// ----------------------------------------------------------
// LI_S Säuretank
// ----------------------------------------------------------
      L     DB1821.DBD 1118; // !!! insert correct SFM !!!
      T     DB2823.DBD  238;

//      SET
//      =     "U082AnID".LI_S.EAlHH

// ----------------------------------------------------------
// CS_S Säuretank
// ----------------------------------------------------------
      L     DB1821.DBD 1118; // !!! insert correct SFM !!!
      T     DB2823.DBD  358;

      SET   ;
      =     DB2823.DBX  261.5;

NETWORK
TITLE =Universal Value

      NOP   0;

// ----------------------------------------------------------
// unv001 Process Status
// ----------------------------------------------------------
// process value to UnV
//      L     0.000000e+000
//      T     "U082UnVD".unv001.ValExt

// ----------------------------------------------------------
// unv002 Universal Value 02
// ----------------------------------------------------------
// process value to UnV
//      L     0.000000e+000
//      T     "U082UnVD".unv002.ValExt

NETWORK
TITLE =Special Input

      NOP   0;

// ----------------------------------------------------------
// LS_LLL_SAEURE Säuretank LS-
// ----------------------------------------------------------
      ON    DB2910.DBX  582.5;
      ON    DB2920.DBX  582.5;
      ON    DB2930.DBX  582.5;
      =     DB2821.DBX   81.4;
      CLR   ;
      =     DB2821.DBX   81.5;

// ----------------------------------------------------------
// LS_HL_SAEURE Säuretank LS+
// ----------------------------------------------------------
      ON    DB2910.DBX  822.5;
      ON    DB2920.DBX  822.5;
      ON    DB2930.DBX  822.5;
      =     DB2821.DBX  141.4;
      SET   ;
      =     DB2821.DBX  141.5;

      SET   ;
      =     DB2821.DBX  140.6;

// ----------------------------------------------------------
// LS_LL_SAEURE Säuretank LS/
// ----------------------------------------------------------
      CLR   ;
//      =     "U082SpID".LS_LL_SAEURE.EAl
      =     DB2821.DBX  201.5;

// ----------------------------------------------------------
// LS_LL_SAEURE_ALT
// ----------------------------------------------------------
      SET   ;
      =     DB2821.DBX  261.4;
      =     DB2821.DBX  261.5;

// ----------------------------------------------------------
// LANG_NEUANSATZ_SAEURE RUECKMELDUNG VON LANG AN TU
// ----------------------------------------------------------
      CLR   ;
//      =     "U082SpID".LANG_NEUANSATZ_SAEURE.EAl
//     =     "U082SpID".LANG_NEUANSATZ_SAEURE.Pre

// ----------------------------------------------------------
// LANG_NACHSCH_SAEURE RUECKMELDUNG VON LANG AN TU
// ----------------------------------------------------------
      CLR   ;
//      =     "U082SpID".LANG_NACHSCH_SAEURE.EAl
//      =     "U082SpID".LANG_NACHSCH_SAEURE.Pre

NETWORK
TITLE =Messages

      NOP   0;

// ----------------------------------------------------------
// msg001 Message 01
// ----------------------------------------------------------
      SET   ;
      R     DB2827.DBX   80.7;
      =     DB2827.DBX   81.4;

      CLR   ;
      =     DB2827.DBX   82.7;

// ----------------------------------------------------------
// msg002 Message 02
// ----------------------------------------------------------
      SET   ;
      R     DB2827.DBX  140.7;
      =     DB2827.DBX  141.4;

      CLR   ;
      =     DB2827.DBX  142.7;

NETWORK
TITLE =Sequence organisation

      CLR   ;
      =     M    122.2;

// SFM supply ----------------------------------------------------------------

// analog value to SFM Säuretank -----------------------
      L     DB2823.DBD  146;
      T     DB1821.DBD  386; // Level

// analog value to SFM Säuretank -----------------------
      L     DB2823.DBD  266;
      T     DB1821.DBD  642; // Conductivity
      T     DB1821.DBD  658; // Conductivity Start Pulse/Pause

// sequencer ----------------------------------------------------------------
      A     DB1823.DBX   43.1;
      S     DB1823.DBX   97.3;

      CALL FC    40 (
           UnitNo                   := #UnitNo);

NETWORK
TITLE =Auto / Manual

      SET   ;
      AN    M    122.2;
      JC    MODE;
      AN    M    120.1;

// assign actuator mode
      AN    M    120.1;
      =     DB2820.DBX  105.4;
      =     DB2820.DBX  185.4;
      =     DB2820.DBX  345.4;
      =     DB2820.DBX  425.4;
      =     DB2820.DBX  585.4;
      =     DB2820.DBX  665.4;
      =     DB2820.DBX  745.4;



MODE: SET   ;

NETWORK
TITLE =RW_SAEURE Rührwerk S1T
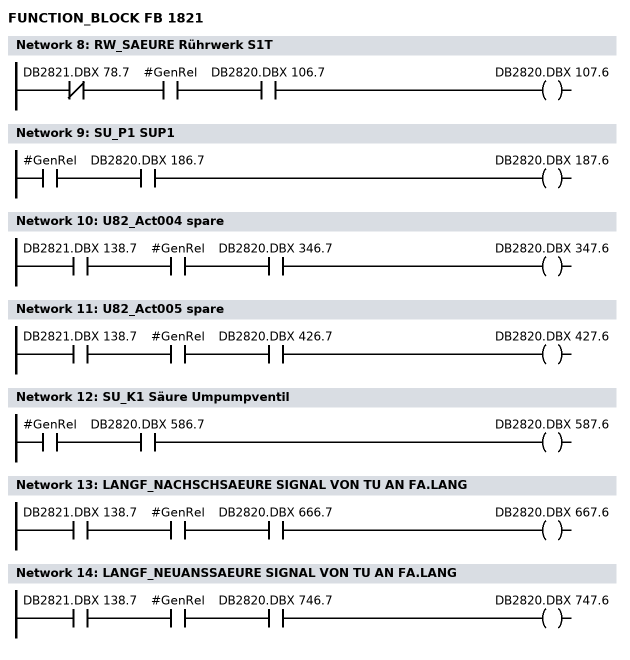

      AN    DB2821.DBX   78.7;
      A     #GenRel;
      A     DB2820.DBX  106.7;
      =     DB2820.DBX  107.6;
NETWORK
TITLE =SU_P1 SUP1

      A     #GenRel;
      A     DB2820.DBX  186.7;
      =     DB2820.DBX  187.6;
NETWORK
TITLE =U82_Act004 spare

      A     DB2821.DBX  138.7;

      A     #GenRel;
      A     DB2820.DBX  346.7;
      =     DB2820.DBX  347.6;
NETWORK
TITLE =U82_Act005 spare

      A     DB2821.DBX  138.7;

      A     #GenRel;
      A     DB2820.DBX  426.7;
      =     DB2820.DBX  427.6;
NETWORK
TITLE =SU_K1 Säure Umpumpventil

      A     #GenRel;
      A     DB2820.DBX  586.7;
      =     DB2820.DBX  587.6;
NETWORK
TITLE =LANGF_NACHSCHSAEURE SIGNAL VON TU AN FA.LANG

      A     DB2821.DBX  138.7;

      A     #GenRel;
      A     DB2820.DBX  666.7;
      =     DB2820.DBX  667.6;
NETWORK
TITLE =LANGF_NEUANSSAEURE SIGNAL VON TU AN FA.LANG

      A     DB2821.DBX  138.7;

      A     #GenRel;
      A     DB2820.DBX  746.7;
      =     DB2820.DBX  747.6;
END_FUNCTION_BLOCK

FUNCTION_BLOCK FB 1830
TITLE =U083: Hot Water Tank
FAMILY : BOTEC_F1
NAME : UniA
VERSION : 2.1


VAR_TEMP
  EStopOK : BOOL ;	//auxiliary flag
  CIP : BOOL ;	//CIP Program Selected
  xTmp : BOOL ;	//Temporary Bool(free for general use)
  UnitNo : INT ;	//unit number
  UnitFB : INT ;	//unit expansion FB number
  rTmp : REAL ;	//Temporary REAL (free for general use)
  iTmp : INT ;	//Temporary INT (free for general use)
  dTmp : DINT ;	//Temporary DINT (free for general use)
END_VAR
BEGIN
NETWORK
TITLE =general

      CLR   ;
      =     #xTmp;
      =     #EStopOK;

      L     DB1830.DBW    0;
      T     #UnitNo;
      L     DB1830.DBW    2;
      T     #UnitFB;

NETWORK
TITLE =analog inputs

      NOP   0;
// LI_HW AnI 001 Niveau Heisswassertank
      CALL FC    24 (
           UnitNo                   := #UnitNo,
           AnIRec                   := DB2833.LI_HW,
           ValPer                   := IW   534);

// HWT_TT01 AnI 002 Temp. HWT
      CALL FC    24 (
           UnitNo                   := #UnitNo,
           AnIRec                   := DB2833.HWT_TT01,
           ValPer                   := IW   536);

// HWT_PIC02 AnI 003
      CALL FC    24 (
           UnitNo                   := #UnitNo,
           AnIRec                   := DB2833.HWT_PIC02,
           ValPer                   := IW   542);

// U83_AnI004 AnI 004 spare
      CALL FC    24 (
           UnitNo                   := #UnitNo,
           AnIRec                   := DB2833.U83_AnI004,
           ValPer                   := IW   236);

// HWT_TT02 AnI 005 Temp. nach Ausdehnungsgefaess
      CALL FC    24 (
           UnitNo                   := #UnitNo,
           AnIRec                   := DB2833.HWT_TT02,
           ValPer                   := IW   538);

// HWT_FT01 AnI 006
      CALL FC    24 (
           UnitNo                   := #UnitNo,
           AnIRec                   := DB2833.HWT_FT01,
           ValPer                   := IW   544);

NETWORK
TITLE =Universal value

      NOP   0;
// unv001 UnV 001 Process Status
      CALL FC    27 (
           UnitNo                   := #UnitNo,
           UnVRec                   := DB2835.unv001,
           ValExt                   := DB2835.DBD  234);

// unv002 UnV 002 Universal Value 02
      CALL FC    27 (
           UnitNo                   := #UnitNo,
           UnVRec                   := DB2835.unv002,
           ValExt                   := DB2835.DBD  362);

NETWORK
TITLE =special inputs

      NOP   0;
// LS_LL_HWT SpI 001 Heißwassertank LS-
      CALL FC    14 (
           UnitNo                   := #UnitNo,
           SpIRec                   := DB2831.LS_LL_HWT,
           SpIBit                   := I     93.4);

// LS_HL_HWT SpI 002 Heißwassertank LS+
      CALL FC    14 (
           UnitNo                   := #UnitNo,
           SpIRec                   := DB2831.LS_HL_HWT,
           SpIBit                   := I     93.2);

// LS_HL_HWA SpI 003 Ausdehnungsgefäß HWT LS+
      CALL FC    14 (
           UnitNo                   := #UnitNo,
           SpIRec                   := DB2831.LS_HL_HWA,
           SpIBit                   := I     93.3);

// SpI4 SpI 004 spare
      CALL FC    14 (
           UnitNo                   := #UnitNo,
           SpIRec                   := DB2831.SpI4,
           SpIBit                   := #xTmp);

// RM_NI_HW_K1 SpI 005
      CALL FC    14 (
           UnitNo                   := #UnitNo,
           SpIRec                   := DB2831.RM_NI_HW_K1,
           SpIBit                   := I     68.4);

// NI_PANEEL_3_NI1 SpI 006 PANEEL3 RV.K2 - HWT
      CALL FC    14 (
           UnitNo                   := #UnitNo,
           SpIRec                   := DB2831.NI_PANEEL_3_NI1,
           SpIBit                   := I     68.0);

// S6_HWP1_HAND_EIN_LAUTO SpI 007 SCHALTER PUMPE HW.P1
      CALL FC    14 (
           UnitNo                   := #UnitNo,
           SpIRec                   := DB2831.S6_HWP1_HAND_EIN_LAUTO,
           SpIBit                   := I     64.3);

NETWORK
TITLE =messages

      NOP   0;
// msg001 Msg 001 Message 01
      CALL FC    16 (
           UnitNo                   := #UnitNo,
           MsgRec                   := DB2837.msg001,
           MsgBit                   := DB2837.DBX   82.7);

// msg002 Msg 002 Message 02
      CALL FC    16 (
           UnitNo                   := #UnitNo,
           MsgRec                   := DB2837.msg002,
           MsgBit                   := DB2837.DBX  142.7);

NETWORK
TITLE =counters

      NOP   0;
// U83_Cnt001 Cnt 001 spare
      CALL FC    25 (
           UnitNo                   := #UnitNo,
           CntRec                   := DB2832.U83_Cnt001,
           Imp                      := DB2832.DBX   99.0);

NETWORK
TITLE =controllers

      NOP   0;
// HWP1_FU PID 001 FU Heisswasserpumpe
      CALL FC    55 (
           UnitNo                   := #UnitNo,
           PIDRec                   := DB2836.HWP1_FU,
           SpExt                    := DB2836.DBD  234,
           PVal                     := DB2836.DBD  254,
           OPer                     := PQW  532);

// RV_Kaltwasser PID 002 Kaltwasser Regelventil HWT
      CALL FC    55 (
           UnitNo                   := #UnitNo,
           PIDRec                   := DB2836.RV_Kaltwasser,
           SpExt                    := DB2836.DBD  414,
           PVal                     := DB2836.DBD  434,
           OPer                     := QW   524);

// U83_PID003 PID 003 spare
      CALL FC    55 (
           UnitNo                   := #UnitNo,
           PIDRec                   := DB2836.U83_PID003,
           SpExt                    := DB2836.DBD  594,
           PVal                     := DB2836.DBD  614,
           OPer                     := QW   232);// S5 ?

NETWORK
TITLE =unit supply

      UC    FB [#UnitFB];

NETWORK
TITLE =HWP1  Heisswasserpumpe Ansteuerung FU
// Act 001
// Box           : LT-CIP
// Input address : I256.5
// Output address: Q256.5
      CALL FC    70 (
           UnitNo                   := #UnitNo,
           ActRec                   := DB2830.HWP1,
           Typ                      := 0,
           FBa                      := #xTmp,
           FBa2                     := #xTmp,
           Out                      := Q    256.5);

NETWORK
TITLE =HWP1_NETZ  Heisswasserpumpe Netzschütz
// Act 002
// Box           : LT-CIP
// Output address: Q256.6
      CALL FC    70 (
           UnitNo                   := #UnitNo,
           ActRec                   := DB2830.HWP1_NETZ,
           Typ                      := 1,
           FBa                      := #xTmp,
           FBa2                     := I    256.5,
           Out                      := Q    256.6);

NETWORK
TITLE =U83_Act003  spare
// Act 003
// Box           :
// Output address: #xTmp
      CALL FC    70 (
           UnitNo                   := #UnitNo,
           ActRec                   := DB2830.U83_Act003,
           Typ                      := 0,
           FBa                      := #xTmp,
           FBa2                     := #xTmp,
           Out                      := #xTmp);

NETWORK
TITLE =U83_Act004  spare
// Act 004
// Box           :
// Output address: #xTmp
      CALL FC    70 (
           UnitNo                   := #UnitNo,
           ActRec                   := DB2830.U83_Act004,
           Typ                      := 0,
           FBa                      := #xTmp,
           FBa2                     := #xTmp,
           Out                      := #xTmp);

NETWORK
TITLE =U83_Act005  spare
// Act 005
// Box           :
// Output address: #xTmp
      CALL FC    70 (
           UnitNo                   := #UnitNo,
           ActRec                   := DB2830.U83_Act005,
           Typ                      := 0,
           FBa                      := #xTmp,
           FBa2                     := #xTmp,
           Out                      := #xTmp);

NETWORK
TITLE =HWT_V1  HWT Abnahmeventil
// Act 007
// Box           : VSRVK1..3
// Input address : I275.6
// Output address: Q275.6
      CALL FC    70 (
           UnitNo                   := #UnitNo,
           ActRec                   := DB2830.HWT_V1,
           Typ                      := 1,
           FBa                      := #xTmp,
           FBa2                     := I    275.6,
           Out                      := Q    275.6);

NETWORK
TITLE =HWT_V2
// Act 009
// Box           : VS-RRA
// Input address : I201.2
// Output address: Q201.2
      CALL FC    70 (
           UnitNo                   := #UnitNo,
           ActRec                   := DB2830.HWT_V2,
           Typ                      := 1,
           FBa                      := #xTmp,
           FBa2                     := I    201.2,
           Out                      := Q    201.2);

NETWORK
TITLE =HWT_V3
// Act 010
// Box           : VS-RRA
// Input address : I201.3
// Output address: Q201.3
      CALL FC    70 (
           UnitNo                   := #UnitNo,
           ActRec                   := DB2830.HWT_V3,
           Typ                      := 1,
           FBa                      := #xTmp,
           FBa2                     := I    201.3,
           Out                      := Q    201.3);

NETWORK
TITLE =HW_WT1_V1  NEU Dampfabsperrung HW-WT1 schließen
// Act 011
// Box           : VSHF9
// Input address : I116.7
// Output address: Q117.0
//      CALL  "Act"
//       UnitNo:=#UnitNo
//       ActRec:="U083ActD".HW_WT1_V1
//       Typ   :=0
//       FBa   :=#xTmp
//       FBa2  :="HW_WT1_V1GSC"
//       Out   :="HW_WT1_V1O"

NETWORK
TITLE =HWT_V4  HWT Luftventil Ausdehnungsgefäß
// Act 012
// Box           : VSRVK1..3
// Input address : I275.7
// Output address: Q275.7
      CALL FC    70 (
           UnitNo                   := #UnitNo,
           ActRec                   := DB2830.HWT_V4,
           Typ                      := 1,
           FBa                      := #xTmp,
           FBa2                     := I    275.7,
           Out                      := Q    275.7);

NETWORK
TITLE =HW_WT1_V1O  NEU Dampfabsperrung HW-WT1 öffnen
// Act 013
// Box           : VSHF9
// Output address: Q116.7

      CALL FC    70 (
           UnitNo                   := #UnitNo,
           ActRec                   := DB2830.HW_WT1_V1O,
           Typ                      := 1,
           FBa                      := #xTmp,
           FBa2                     := I    116.7,
           Out                      := Q    117.0);

END_FUNCTION_BLOCK

FUNCTION_BLOCK FB 1831
TITLE =U083: Hot Water Tank
FAMILY : BOTEC_F1
NAME : UniE
VERSION : 1.2


VAR_TEMP
  CIP : BOOL ;	//CIP active
  UNIM : BOOL ;	//Unit Not In Maintenance
  GenRel : BOOL ;	//general OK (emergency and maintenance OK)
  EStopOK : BOOL ;	//emergency OK
  UnitNo : INT ;	//unit number
  xTmp : BOOL ;	//Temporary Bool
  iTmp : INT ;	//Temporary INT
  rTmp : REAL ;	//Temporary REAL
  dTmp : DINT ;	//Temporary DINT (free for general use)
  RetValInt : INT ;	//return value
END_VAR
BEGIN
NETWORK
TITLE =General

      SET   ;
// Simulation ---------------------------------------------------------------
      A     DB1831.DBX 1357.7;
      CC    FB  1839; // "U083Sim"
      A     DB1831.DBX   17.3;
      =     DB1831.DBX 1357.7; //Help bit for simulation

// get unit number ----------------------------------------------------------
      L     DB1830.DBW    0;
      T     #UnitNo;

// CIP ----------------------------------------------------------------------
      L     DB1831.DBD   54;
      L     0;
      <D    ;
      =     #CIP;

// emergency OK -------------------------------------------------------------
      A     DB1835.DBX   27.0; //Emergency Stop OK
      =     #EStopOK;

// Write Unit in Maintenance ------------------------------------------------

      AN    DB1831.DBX   69.7;
      =     #UNIM;

// emergency and maintenance OK ---------------------------------------------
      A     #EStopOK;
      A     #UNIM;
      =     #GenRel;

// communication ------------------------------------------------------------
      UC    FB  1835; // U083Com

NETWORK
TITLE =Analog Inputs

      NOP   0;

// ----------------------------------------------------------
// LI_HW Niveau Heisswassertank
// ----------------------------------------------------------
      L     DB1831.DBD 1118; // !!! insert correct SFM !!!
      T     DB2833.DBD  238;

//      SET
//      =     "U083AnID".LI_HW.EAlHH

// ----------------------------------------------------------
// HWT_TT01 Temp. HWT
// ----------------------------------------------------------
      L     DB1831.DBD 1118; // !!! insert correct SFM !!!
      T     DB2833.DBD  358;

      SET   ;
      =     DB2833.DBX  261.5;

// ----------------------------------------------------------
// HWT_PIC02
// ----------------------------------------------------------
      L     DB1831.DBD 1118; // !!! insert correct SFM !!!
      T     DB2833.DBD  478;

      SET   ;
      =     DB2833.DBX  381.5;

// ----------------------------------------------------------
// U83_AnI004
// ----------------------------------------------------------
      L     DB1831.DBD 1118; // !!! insert correct SFM !!!
      T     DB2833.DBD  598;

      SET   ;
      =     DB2833.DBX  501.5;

// ----------------------------------------------------------
// HWT_TT02 Temp. nach Ausdehnungsgefaess
// ----------------------------------------------------------
      L     DB1831.DBD 1118; // !!! insert correct SFM !!!
      T     DB2833.DBD  718;

      SET   ;
      =     DB2833.DBX  621.5;

// ----------------------------------------------------------
// HWT_FT01
// ----------------------------------------------------------
      L     DB1831.DBD 1118; // !!! insert correct SFM !!!
      T     DB2833.DBD  838;

      SET   ;
      =     DB2833.DBX  741.5;

NETWORK
TITLE =Universal Value

      NOP   0;

// ----------------------------------------------------------
// unv001 Process Status
// ----------------------------------------------------------
// process value to UnV
//      L     0.000000e+000
//      T     "U083UnVD".unv001.ValExt

// ----------------------------------------------------------
// unv002 Universal Value 02
// ----------------------------------------------------------
// process value to UnV
//      L     0.000000e+000
//      T     "U083UnVD".unv002.ValExt

NETWORK
TITLE =Special Input

      NOP   0;

// ----------------------------------------------------------
// LS_LL_HWT Heißwassertank LS-
// ----------------------------------------------------------
      ON    DB2910.DBX  502.5;
      ON    DB2920.DBX  502.5;
      ON    DB2930.DBX  502.5;
      =     DB2831.DBX   81.4;
      CLR   ;
      =     DB2831.DBX   81.5;

// ----------------------------------------------------------
// LS_HL_HWT Heißwassertank LS+
// ----------------------------------------------------------
      ON    DB2930.DBX  902.5;
      ON    DB2920.DBX  902.5;
      ON    DB2910.DBX  902.5;
      =     DB2831.DBX  141.4;
      SET   ;
      =     DB2831.DBX  141.5;

      CLR   ;
      =     DB2831.DBX  140.6;

// ----------------------------------------------------------
// LS_HL_HWA Ausdehnungsgefäß HWT LS+
// ----------------------------------------------------------
      A     DB2830.DBX  982.6;
      O     DB2830.DBX  182.6;
      =     DB2831.DBX  201.4;
      SET   ;
      =     DB2831.DBX  201.5;

// ----------------------------------------------------------
// SpI4 spare
// ----------------------------------------------------------
//      SET
//      =     "U083SpID".SpI4.EAl
//      =     "U083SpID".SpI4.Pre

// ----------------------------------------------------------
// RM_NI_HW_K1
// ----------------------------------------------------------
      SET   ;
      =     DB2831.DBX  321.4;
      =     DB2831.DBX  321.5;

// ----------------------------------------------------------
// NI_PANEEL_3_NI1 PANEEL3 RV.K2 - HWT
// ----------------------------------------------------------
      SET   ;
      =     DB2831.DBX  381.4;
      CLR   ;
      =     DB2831.DBX  381.5;

// ----------------------------------------------------------
// S6_HWP1_HAND_EIN_LAUTO SCHALTER PUMPE HW.P1
// ----------------------------------------------------------
//      CLR
//      =     "U083SpID".S6_HWP1_HAND_EIN_LAUTO.EAl
//      =     "U083SpID".S6_HWP1_HAND_EIN_LAUTO.Pre

NETWORK
TITLE =Messages

      NOP   0;

// ----------------------------------------------------------
// msg001 Message 01
// ----------------------------------------------------------
      SET   ;
      R     DB2837.DBX   80.7;
      =     DB2837.DBX   81.4;

      CLR   ;
      =     DB2837.DBX   82.7;

// ----------------------------------------------------------
// msg002 Message 02
// ----------------------------------------------------------
      SET   ;
      R     DB2837.DBX  140.7;
      =     DB2837.DBX  141.4;

      CLR   ;
      =     DB2837.DBX  142.7;

NETWORK
TITLE =Counters

      NOP   0;

// ----------------------------------------------------------
// U83_Cnt001 spare
// ----------------------------------------------------------
//A     "U083ActD".Act.VOn // !!! insert correct Act !!!
      CLR   ;
      =     DB2832.DBX  103.5;

//AN    "U083ActD".Act.VOff // !!! insert correct Act !!!
//A     "U083SpID".SpI.Sig // !!! insert correct SpI !!!
      CLR   ;
      =     DB2832.DBX   99.0;

NETWORK
TITLE =PID controller
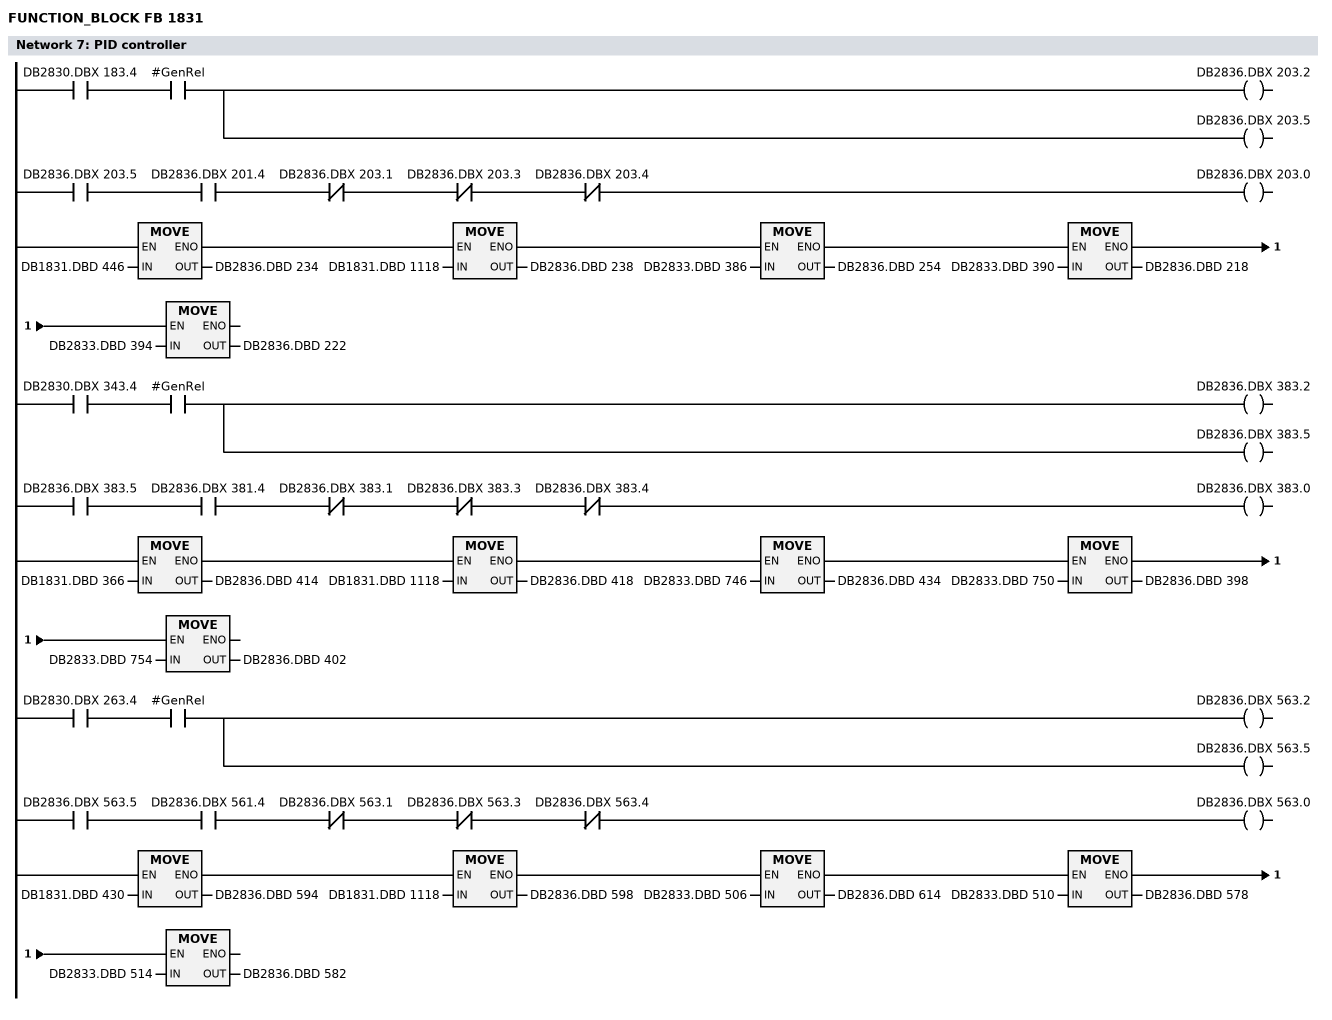

      NOP   0;

// ----------------------------------------------------------
// HWP1_FU FU Heisswasserpumpe
// ----------------------------------------------------------
// starting value -----------------------
      A     DB2830.DBX  183.4;
      A     #GenRel;
      =     DB2836.DBX  203.2;
      =     DB2836.DBX  203.5;

// enable alarm -------------------------
      A     DB2836.DBX  203.5;
      A     DB2836.DBX  201.4;
      AN    DB2836.DBX  203.1;
      AN    DB2836.DBX  203.3;
      AN    DB2836.DBX  203.4;
      =     DB2836.DBX  203.0;

// setpoint to controller ---------------
      L     DB1831.DBD  446; // Pressure
      T     DB2836.DBD  234;

// static value to controller ----------
      L     DB1831.DBD 1118; // !!! insert correct SFM !!!
      T     DB2836.DBD  238;

// process value to controller ----------
      L     DB2833.DBD  386;
      T     DB2836.DBD  254;

// low/high value to controller ---------
      L     DB2833.DBD  390; // Pressure
      T     DB2836.DBD  218;

      L     DB2833.DBD  394; // Pressure
      T     DB2836.DBD  222;

// ----------------------------------------------------------
// RV_Kaltwasser Kaltwasser Regelventil HWT
// ----------------------------------------------------------
// starting value -----------------------
      A     DB2830.DBX  343.4;
      A     #GenRel;
      =     DB2836.DBX  383.2;
      =     DB2836.DBX  383.5;

// enable alarm -------------------------
      A     DB2836.DBX  383.5;
      A     DB2836.DBX  381.4;
      AN    DB2836.DBX  383.1;
      AN    DB2836.DBX  383.3;
      AN    DB2836.DBX  383.4;
      =     DB2836.DBX  383.0;

// setpoint to controller ---------------
      L     DB1831.DBD  366; // Flow Water Inlet
      T     DB2836.DBD  414;

// static value to controller ----------
      L     DB1831.DBD 1118; // !!! insert correct SFM !!!
      T     DB2836.DBD  418;

// process value to controller ----------
      L     DB2833.DBD  746; // Flow Water
      T     DB2836.DBD  434;

// low/high value to controller ---------
      L     DB2833.DBD  750; // Flow Water
      T     DB2836.DBD  398;

      L     DB2833.DBD  754; // Flow Water
      T     DB2836.DBD  402;

// ----------------------------------------------------------
// U83_PID003 spare
// ----------------------------------------------------------
// starting value -----------------------
      A     DB2830.DBX  263.4;
      A     #GenRel;
      =     DB2836.DBX  563.2;
      =     DB2836.DBX  563.5;

// enable alarm -------------------------
      A     DB2836.DBX  563.5;
      A     DB2836.DBX  561.4;
      AN    DB2836.DBX  563.1;
      AN    DB2836.DBX  563.3;
      AN    DB2836.DBX  563.4;
      =     DB2836.DBX  563.0;

// setpoint to controller ---------------
      L     DB1831.DBD  430; // Temperature Heater
      T     DB2836.DBD  594;

// static value to controller ----------
      L     DB1831.DBD 1118; // !!! insert correct SFM !!!
      T     DB2836.DBD  598;

// process value to controller ----------
      L     DB2833.DBD  506; // Temp. After Heater
      T     DB2836.DBD  614;

// low/high value to controller ---------
      L     DB2833.DBD  510; // Temp. After Heater
      T     DB2836.DBD  578;

      L     DB2833.DBD  514; // Temp. After Heater
      T     DB2836.DBD  582;

NETWORK
TITLE =Sequence organisation

      CLR   ;
      =     M    122.2;

// SFM supply ----------------------------------------------------------------
// analog value to SFM Niveau Heisswassertank -----------------------
      L     DB2833.DBD  146;
      T     DB1831.DBD  386; // Level

// analog value to SFM Temp. HWT -----------------------
      L     DB2833.DBD  266;
      T     DB1831.DBD  402; // Temperature

// analog value to SFM  -----------------------
      L     DB2833.DBD  386;
      T     DB1831.DBD  450; // Pressure

// analog value to SFM Temp. nach Ausdehnungsgefaess -----------------------
      L     DB2833.DBD  506;
      T     DB1831.DBD  434; // Temperature Heater

// analog value to SFM  -----------------------
      L     DB2833.DBD  746;
      T     DB1831.DBD  370; // Flow Water Inlet

// sequencer ----------------------------------------------------------------
      A     DB1833.DBX   43.1;
      S     DB1833.DBX   97.3;

      CALL FC    40 (
           UnitNo                   := #UnitNo);

NETWORK
TITLE =Auto / Manual

      SET   ;
      AN    M    122.2;
      JC    MODE;
      AN    M    120.1;

// assign actuator mode
      AN    M    120.1;
      =     DB2830.DBX  105.4;
      =     DB2830.DBX  185.4;
      =     DB2830.DBX  265.4;
      =     DB2830.DBX  345.4;
      =     DB2830.DBX  425.4;
      =     DB2830.DBX  585.4;
      =     DB2830.DBX  745.4;
      =     DB2830.DBX  825.4;
      =     DB2830.DBX  905.4;
      =     DB2830.DBX  985.4;
      =     DB2830.DBX 1065.4;

// assign PID mode
      S     DB2836.DBX  201.4;
      S     DB2836.DBX  201.5;
      S     DB2836.DBX  381.4;
      S     DB2836.DBX  381.5;
      S     DB2836.DBX  561.4;
      S     DB2836.DBX  561.5;



MODE: SET   ;

NETWORK
TITLE =HWP1 Heisswasserpumpe Ansteuerung FU
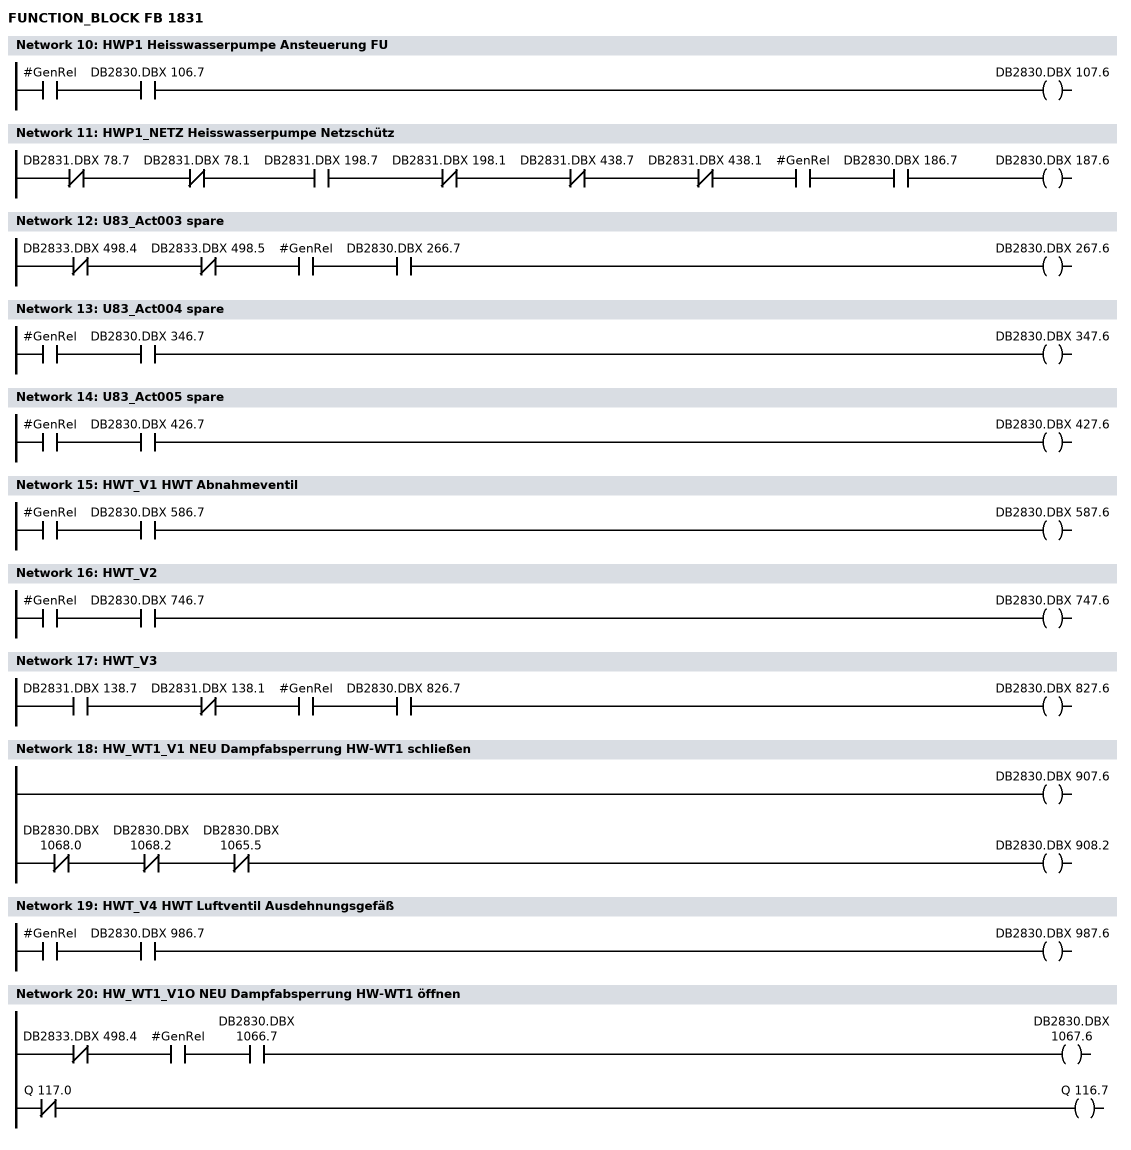

      A     #GenRel;
      A     DB2830.DBX  106.7;
      =     DB2830.DBX  107.6;
NETWORK
TITLE =HWP1_NETZ Heisswasserpumpe Netzschütz

      AN    DB2831.DBX   78.7;
      AN    DB2831.DBX   78.1;

      A     DB2831.DBX  198.7;
      AN    DB2831.DBX  198.1;

      AN    DB2831.DBX  438.7;
      AN    DB2831.DBX  438.1;

      A     #GenRel;
      A     DB2830.DBX  186.7;
      =     DB2830.DBX  187.6;
NETWORK
TITLE =U83_Act003 spare

      AN    DB2833.DBX  498.4;
      AN    DB2833.DBX  498.5;

      A     #GenRel;
      A     DB2830.DBX  266.7;
      =     DB2830.DBX  267.6;

NETWORK
TITLE =U83_Act004 spare

      A     #GenRel;
      A     DB2830.DBX  346.7;
      =     DB2830.DBX  347.6;

NETWORK
TITLE =U83_Act005 spare

      A     #GenRel;
      A     DB2830.DBX  426.7;
      =     DB2830.DBX  427.6;

NETWORK
TITLE =HWT_V1 HWT Abnahmeventil

      A     #GenRel;
      A     DB2830.DBX  586.7;
      =     DB2830.DBX  587.6;
NETWORK
TITLE =HWT_V2

      A     #GenRel;
      A     DB2830.DBX  746.7;
      =     DB2830.DBX  747.6;
NETWORK
TITLE =HWT_V3

      A     DB2831.DBX  138.7;
      AN    DB2831.DBX  138.1;

      A     #GenRel;
      A     DB2830.DBX  826.7;
      =     DB2830.DBX  827.6;
NETWORK
TITLE =HW_WT1_V1 NEU Dampfabsperrung HW-WT1 schließen

      SET   ;
      =     DB2830.DBX  907.6;

      AN    DB2830.DBX 1068.0;
      AN    DB2830.DBX 1068.2;
      AN    DB2830.DBX 1065.5;
      =     DB2830.DBX  908.2;
NETWORK
TITLE =HWT_V4 HWT Luftventil Ausdehnungsgefäß

      A     #GenRel;
      A     DB2830.DBX  986.7;
      =     DB2830.DBX  987.6;
NETWORK
TITLE =HW_WT1_V1O NEU Dampfabsperrung HW-WT1 öffnen

      AN    DB2833.DBX  498.4;
      A     #GenRel;
      A     DB2830.DBX 1066.7;
      =     DB2830.DBX 1067.6;


      AN    Q    117.0;
//     =       Q    117.0
      =     Q    116.7;
END_FUNCTION_BLOCK

FUNCTION_BLOCK FB 1840
TITLE =U084: Fresh Water Tank
FAMILY : BOTEC_F1
NAME : UniA
VERSION : 2.1


VAR_TEMP
  EStopOK : BOOL ;	//auxiliary flag
  CIP : BOOL ;	//CIP Program Selected
  xTmp : BOOL ;	//Temporary Bool(free for general use)
  UnitNo : INT ;	//unit number
  UnitFB : INT ;	//unit expansion FB number
  rTmp : REAL ;	//Temporary REAL (free for general use)
  iTmp : INT ;	//Temporary INT (free for general use)
  dTmp : DINT ;	//Temporary DINT (free for general use)
END_VAR
BEGIN
NETWORK
TITLE =general

      CLR   ;
      =     #xTmp;
      =     #EStopOK;

      L     DB1840.DBW    0;
      T     #UnitNo;
      L     DB1840.DBW    2;
      T     #UnitFB;

NETWORK
TITLE =analog inputs

      NOP   0;
// LI_FW AnI 001 Frischwassertank
      CALL FC    24 (
           UnitNo                   := #UnitNo,
           AnIRec                   := DB2843.LI_FW,
           ValPer                   := IW   568);

NETWORK
TITLE =Universal value

      NOP   0;
// unv001 UnV 001 Process Status
      CALL FC    27 (
           UnitNo                   := #UnitNo,
           UnVRec                   := DB2845.unv001,
           ValExt                   := DB2845.DBD  234);

// unv002 UnV 002 Universal Value 02
      CALL FC    27 (
           UnitNo                   := #UnitNo,
           UnVRec                   := DB2845.unv002,
           ValExt                   := DB2845.DBD  362);

NETWORK
TITLE =special inputs


// LS_LLL_FW_ALT SpI 001 spare
      CALL FC    14 (
           UnitNo                   := #UnitNo,
           SpIRec                   := DB2841.LS_LLL_FW_ALT,
           SpIBit                   := I     42.5);

// LS_HL_FW_ALT SpI 002 spare
      CALL FC    14 (
           UnitNo                   := #UnitNo,
           SpIRec                   := DB2841.LS_HL_FW_ALT,
           SpIBit                   := I     42.3);

// LS_LL_FW_ALT SpI 003 spare
      CALL FC    14 (
           UnitNo                   := #UnitNo,
           SpIRec                   := DB2841.LS_LL_FW_ALT,
           SpIBit                   := I     42.4);

// RM_NI_FW_K1 SpI 005
      CALL FC    14 (
           UnitNo                   := #UnitNo,
           SpIRec                   := DB2841.RM_NI_FW_K1,
           SpIBit                   := I     68.5);

// NI_PANEEL_3_NI2 SpI 006 PANEEL3 RV.K2 - FWT
      CALL FC    14 (
           UnitNo                   := #UnitNo,
           SpIRec                   := DB2841.NI_PANEEL_3_NI2,
           SpIBit                   := I     68.1);

// LANG_NEUANSATZ_OXONIA SpI 007 RUECKMELDUNG VON LANG AN TU
      CALL FC    14 (
           UnitNo                   := #UnitNo,
           SpIRec                   := DB2841.LANG_NEUANSATZ_OXONIA,
           SpIBit                   := I     40.2);

// LANG_NACHSCH_OXONIA SpI 008 RUECKMELDUNG VON LANG AN TU
      CALL FC    14 (
           UnitNo                   := #UnitNo,
           SpIRec                   := DB2841.LANG_NACHSCH_OXONIA,
           SpIBit                   := I     40.6);

      NOP   0;
// LS_LLL_FW_NEU SpI 010 Frischwassertank LS-
//      CALL  "SI1"
//       UnitNo:=#UnitNo
//       SpIRec:="U084SpID".LS_LLL_FW_NEU
//       SpIBit:="LS_LLL_FW_NEU"

// LS_HL_FW_NEU SpI 011 Frischwassertank LS+
//      CALL  "SI1"
//       UnitNo:=#UnitNo
//       SpIRec:="U084SpID".LS_HL_FW_NEU
//       SpIBit:="LS_HL_FW_NEU"

// LS_LL_FW_NEU SpI 012 Frischwassertank LS/
//      CALL  "SI1"
//       UnitNo:=#UnitNo
//       SpIRec:="U084SpID".LS_LL_FW_NEU
//       SpIBit:="LS_LL_FW_NEU"



// RM_NI_FW_P1_K1 SpI 015
      CALL FC    14 (
           UnitNo                   := #UnitNo,
           SpIRec                   := DB2841.RM_NI_FW_P1_K1,
           SpIBit                   := I     61.5);

NETWORK
TITLE =messages

      NOP   0;
// msg001 Msg 001 Message 01
      CALL FC    16 (
           UnitNo                   := #UnitNo,
           MsgRec                   := DB2847.msg001,
           MsgBit                   := DB2847.DBX   82.7);

// msg002 Msg 002 Message 02
      CALL FC    16 (
           UnitNo                   := #UnitNo,
           MsgRec                   := DB2847.msg002,
           MsgBit                   := DB2847.DBX  142.7);

NETWORK
TITLE =unit supply

      UC    FB [#UnitFB];

NETWORK
TITLE =FW_V4  Frischwasserbehälter Befüllventil
// Act 002
// Box           : VSRVK1..3
// Input address : I273.4
// Output address: Q273.4
      CALL FC    70 (
           UnitNo                   := #UnitNo,
           ActRec                   := DB2840.FW_V4,
           Typ                      := 1,
           FBa                      := #xTmp,
           FBa2                     := I    273.4,
           Out                      := Q    273.4);

NETWORK
TITLE =LANGF_NACHSCHOXONIA  SIGNAL VON TU AN FA.LANG
// Act 008
// Box           : S8 U8.2
// Output address: Q43.2
      CALL FC    70 (
           UnitNo                   := #UnitNo,
           ActRec                   := DB2840.LANGF_NACHSCHOXONIA,
           Typ                      := 0,
           FBa                      := #xTmp,
           FBa2                     := #xTmp,
           Out                      := Q     43.2);

NETWORK
TITLE =LANGF_NEUANSOXONIA  SIGNAL VON TU AN FA.LANG
// Act 009
// Box           : S8 U8.2
// Output address: Q43.5
      CALL FC    70 (
           UnitNo                   := #UnitNo,
           ActRec                   := DB2840.LANGF_NEUANSOXONIA,
           Typ                      := 0,
           FBa                      := #xTmp,
           FBa2                     := #xTmp,
           Out                      := Q     43.5);

END_FUNCTION_BLOCK

FUNCTION_BLOCK FB 1841
TITLE =U084: Fresh Water Tank
FAMILY : BOTEC_F1
NAME : UniE
VERSION : 1.2


VAR_TEMP
  CIP : BOOL ;	//CIP active
  UNIM : BOOL ;	//Unit Not In Maintenance
  GenRel : BOOL ;	//general OK (emergency and maintenance OK)
  EStopOK : BOOL ;	//emergency OK
  UnitNo : INT ;	//unit number
  xTmp : BOOL ;	//Temporary Bool
  iTmp : INT ;	//Temporary INT
  rTmp : REAL ;	//Temporary REAL
  dTmp : DINT ;	//Temporary DINT (free for general use)
  RetValInt : INT ;	//return value
END_VAR
BEGIN
NETWORK
TITLE =General

      SET   ;
// Simulation ---------------------------------------------------------------
      A     DB1841.DBX 1357.7;
      CC    FB  1849; // "U084Sim"
      A     DB1841.DBX   17.3;
      =     DB1841.DBX 1357.7; //Help bit for simulation

// get unit number ----------------------------------------------------------
      L     DB1840.DBW    0;
      T     #UnitNo;

// CIP ----------------------------------------------------------------------
      L     DB1841.DBD   54;
      L     0;
      <D    ;
      =     #CIP;

// emergency OK -------------------------------------------------------------
      A     DB1845.DBX   27.0; //Emergency Stop OK
      =     #EStopOK;

// Write Unit in Maintenance ------------------------------------------------

      AN    DB1841.DBX   69.7;
      =     #UNIM;

// emergency and maintenance OK ---------------------------------------------
      A     #EStopOK;
      A     #UNIM;
      =     #GenRel;

// communication ------------------------------------------------------------
      UC    FB  1845; // U084Com

NETWORK
TITLE =Analog Inputs

      NOP   0;

// ----------------------------------------------------------
// LI_FW Frischwassertank
// ----------------------------------------------------------
      L     DB1841.DBD 1118; // !!! insert correct SFM !!!
      T     DB2843.DBD  238;

//      SET
//      =     "U084AnID".LI_FW.EAlHH

NETWORK
TITLE =Universal Value

      NOP   0;

// ----------------------------------------------------------
// unv001 Process Status
// ----------------------------------------------------------
// process value to UnV
//      L     0.000000e+000
//      T     "U084UnVD".unv001.ValExt

// ----------------------------------------------------------
// unv002 Universal Value 02
// ----------------------------------------------------------
// process value to UnV
//      L     0.000000e+000
//      T     "U084UnVD".unv002.ValExt

NETWORK
TITLE =Special Input

      NOP   0;

// ----------------------------------------------------------
// LS_LLL_FW_NEU Frischwassertank LS-
// ----------------------------------------------------------
      A     DB2910.DBX  422.6;
      O     DB2920.DBX  422.6;
      O     DB2930.DBX  422.6;
      ON    DB2841.DBX  318.7;
      =     DB2841.DBX   81.4;
      CLR   ;
      =     DB2841.DBX   81.5;

// ----------------------------------------------------------
// LS_HL_FW_NEU Frischwassertank LS+
// ----------------------------------------------------------
      AN    DB2840.DBX  182.5;
      =     DB2841.DBX  141.4;
      =     DB2841.DBX  141.5;

      CLR   ;
      =     DB2841.DBX  140.6;

// ----------------------------------------------------------
// LS_LL_FW_NEU Frischwassertank LS/
// ----------------------------------------------------------
      CLR   ;
//      =     "U084SpID".LS_LL_FW_NEU.EAl
      =     DB2841.DBX  201.5;

// ----------------------------------------------------------
// RM_NI_FW_K1
// ----------------------------------------------------------
      SET   ;
//      =     "U084SpID".RM_NI_FW_K1.EAl
      =     DB2841.DBX  321.5;

// ----------------------------------------------------------
// NI_PANEEL_3_NI2 PANEEL3 RV.K2 - FWT
// ----------------------------------------------------------
      SET   ;
//      =     "U084SpID".NI_PANEEL_3_NI2.EAl
      =     DB2841.DBX  381.5;

// ----------------------------------------------------------
// LANG_NEUANSATZ_OXONIA RUECKMELDUNG VON LANG AN TU
// ----------------------------------------------------------
      CLR   ;
//      =     "U084SpID".LANG_NEUANSATZ_OXONIA.EAl
//      =     "U084SpID".LANG_NEUANSATZ_OXONIA.Pre

// ----------------------------------------------------------
// LANG_NACHSCH_OXONIA RUECKMELDUNG VON LANG AN TU
// ----------------------------------------------------------
      CLR   ;
//      =     "U084SpID".LANG_NACHSCH_OXONIA.EAl
//      =     "U084SpID".LANG_NACHSCH_OXONIA.Pre

// ----------------------------------------------------------
// LS_LLL_FW_ALT
// ----------------------------------------------------------
      CLR   ;
      =     DB2841.DBX  621.4;
      =     DB2841.DBX  621.5;

// ----------------------------------------------------------
// LS_HL_FW_ALT
// ----------------------------------------------------------
      CLR   ;
      =     DB2841.DBX  681.4;
      =     DB2841.DBX  681.5;

// ----------------------------------------------------------
// LS_LL_FW_ALT
// ----------------------------------------------------------
      CLR   ;
      =     DB2841.DBX  741.4;
      =     DB2841.DBX  741.5;

// ----------------------------------------------------------
// RM_NI_FW_P1_K1
// ----------------------------------------------------------
      CLR   ;
//      =     "U084SpID".RM_NI_FW_P1_K1.EAl
      =     DB2841.DBX  921.5;

NETWORK
TITLE =Messages

      NOP   0;

// ----------------------------------------------------------
// msg001 Message 01
// ----------------------------------------------------------
      SET   ;
      R     DB2847.DBX   80.7;
      =     DB2847.DBX   81.4;

      CLR   ;
      =     DB2847.DBX   82.7;

// ----------------------------------------------------------
// msg002 Message 02
// ----------------------------------------------------------
      SET   ;
      R     DB2847.DBX  140.7;
      =     DB2847.DBX  141.4;

      CLR   ;
      =     DB2847.DBX  142.7;

NETWORK
TITLE =Sequence organisation

      CLR   ;
      =     M    122.2;

// SFM supply ----------------------------------------------------------------

// analog value to SFM Frischwassertank -----------------------
      L     DB2843.DBD  146;
      T     DB1841.DBD  386; // Level

// sequencer ----------------------------------------------------------------
      A     DB1843.DBX   43.1;
      S     DB1843.DBX   97.3;

      CALL FC    40 (
           UnitNo                   := #UnitNo);

NETWORK
TITLE =Auto / Manual

      SET   ;
      AN    M    122.2;
      JC    MODE;
      AN    M    120.1;

// assign actuator mode
      AN    M    120.1;
      =     DB2840.DBX  185.4;
      =     DB2840.DBX  665.4;
      =     DB2840.DBX  745.4;



MODE: SET   ;

NETWORK
TITLE =FW_V4 Frischwasserbehälter Befüllventil
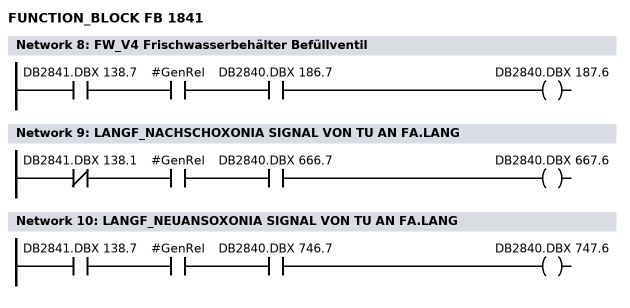

      A     DB2841.DBX  138.7;

      A     #GenRel;
      A     DB2840.DBX  186.7;
      =     DB2840.DBX  187.6;
NETWORK
TITLE =LANGF_NACHSCHOXONIA SIGNAL VON TU AN FA.LANG

      AN    DB2841.DBX  138.1;

      A     #GenRel;
      A     DB2840.DBX  666.7;
      =     DB2840.DBX  667.6;
NETWORK
TITLE =LANGF_NEUANSOXONIA SIGNAL VON TU AN FA.LANG

      A     DB2841.DBX  138.7;

      A     #GenRel;
      A     DB2840.DBX  746.7;
      =     DB2840.DBX  747.6;
END_FUNCTION_BLOCK

FUNCTION_BLOCK FB 1910
TITLE =U091: CIP Line 1
FAMILY : BOTEC_F1
NAME : UniA
VERSION : 2.1


VAR_TEMP
  EStopOK : BOOL ;	//auxiliary flag
  CIP : BOOL ;	//CIP Program Selected
  xTmp : BOOL ;	//Temporary Bool(free for general use)
  UnitNo : INT ;	//unit number
  UnitFB : INT ;	//unit expansion FB number
  rTmp : REAL ;	//Temporary REAL (free for general use)
  iTmp : INT ;	//Temporary INT (free for general use)
  dTmp : DINT ;	//Temporary DINT (free for general use)
END_VAR
BEGIN
NETWORK
TITLE =general

      CLR   ;
      =     #xTmp;
      =     #EStopOK;

      L     DB1910.DBW    0;
      T     #UnitNo;
      L     DB1910.DBW    2;
      T     #UnitFB;

NETWORK
TITLE =analog inputs

      NOP   0;
// RV1T1 AnI 001 Regler 2 RV 1 Temperatur 1
      CALL FC    24 (
           UnitNo                   := #UnitNo,
           AnIRec                   := DB2913.RV1T1,
           ValPer                   := IW   224);

// TI_RR1 AnI 002 Temperatur CIP Rücklauf 1
      CALL FC    24 (
           UnitNo                   := #UnitNo,
           AnIRec                   := DB2913.TI_RR1,
           ValPer                   := IW   134);

// CS_RR1 AnI 003 Messbereich ist umschaltber
      CALL FC    24 (
           UnitNo                   := #UnitNo,
           AnIRec                   := DB2913.CS_RR1,
           ValPer                   := IW   140);

// FIT_RV1 AnI 004 Flow CIP Kreislauf 1
      CALL FC    24 (
           UnitNo                   := #UnitNo,
           AnIRec                   := DB2913.FIT_RV1,
           ValPer                   := IW   128);

NETWORK
TITLE =Universal value

      NOP   0;
// unv001 UnV 001 Process Status
      CALL FC    27 (
           UnitNo                   := #UnitNo,
           UnVRec                   := DB2915.unv001,
           ValExt                   := DB2915.DBD  234);

// unv002 UnV 002 Universal Value 02
      CALL FC    27 (
           UnitNo                   := #UnitNo,
           UnVRec                   := DB2915.unv002,
           ValExt                   := DB2915.DBD  362);

NETWORK
TITLE =special inputs

      NOP   0;
// FS_RR1_NEU SpI 001
      CALL FC    14 (
           UnitNo                   := #UnitNo,
           SpIRec                   := DB2911.FS_RR1_NEU,
           SpIBit                   := I     94.0);

// IDM_IMPULSE_RV_1FQS SpI 002 DURCHFLUSSMESSUNG KREISLAUF 1
      CALL FC    14 (
           UnitNo                   := #UnitNo,
           SpIRec                   := DB2911.IDM_IMPULSE_RV_1FQS,
           SpIBit                   := I      0.0);

NETWORK
TITLE =messages

      NOP   0;
// msg001 Msg 001 Message 01
      CALL FC    16 (
           UnitNo                   := #UnitNo,
           MsgRec                   := DB2917.msg001,
           MsgBit                   := DB2917.DBX   82.7);

// msg002 Msg 002 Message 02
      CALL FC    16 (
           UnitNo                   := #UnitNo,
           MsgRec                   := DB2917.msg002,
           MsgBit                   := DB2917.DBX  142.7);

NETWORK
TITLE =counters

      NOP   0;
// IDM_IMPULSE_RV_1FQI Cnt 002 DURCHFLUSSMESSUNG KREISLAUF 1 (U91)
      CALL FC    25 (
           UnitNo                   := #UnitNo,
           CntRec                   := DB2912.IDM_IMPULSE_RV_1FQI,
           Imp                      := DB2912.DBX  179.0);

NETWORK
TITLE =controllers

      NOP   0;
// RV1RV PID 001 CIP 1
      CALL FC    55 (
           UnitNo                   := #UnitNo,
           PIDRec                   := DB2916.RV1RV,
           SpExt                    := DB2916.DBD  234,
           PVal                     := DB2916.DBD  254,
           OPer                     := QW   224);

NETWORK
TITLE =unit supply

      UC    FB [#UnitFB];

NETWORK
TITLE =RV_P1  Reinigungsvorlaufpumpe Kreis 1
// Act 001
// Box           : LT-CIP
// Input address : I256.0
// Output address: Q256.0
      CALL FC    70 (
           UnitNo                   := #UnitNo,
           ActRec                   := DB2910.RV_P1,
           Typ                      := 3,
           FBa                      := I    256.0,
           FBa2                     := #xTmp,
           Out                      := Q    256.0);

NETWORK
TITLE =RV1_RV  Regelventil CIP 1
// Act 004
// Box           :
// Output address: #DummyBool
      CALL FC    70 (
           UnitNo                   := #UnitNo,
           ActRec                   := DB2910.RV1_RV,
           Typ                      := 0,
           FBa                      := #xTmp,
           FBa2                     := #xTmp,
           Out                      := Q     14.1);

NETWORK
TITLE =FW_V1  Frischwasservorlaufventil Kreis 1
// Act 005
// Box           : VSRVK1..3
// Input address : I273.1
// Output address: Q273.1
      CALL FC    70 (
           UnitNo                   := #UnitNo,
           ActRec                   := DB2910.FW_V1,
           Typ                      := 1,
           FBa                      := #xTmp,
           FBa2                     := I    273.1,
           Out                      := Q    273.1);

NETWORK
TITLE =HW_V1  Heisswasservorlaufventil Kreis 1
// Act 006
// Box           : VSRVK1..3
// Input address : I274.6
// Output address: Q274.6
      CALL FC    70 (
           UnitNo                   := #UnitNo,
           ActRec                   := DB2910.HW_V1,
           Typ                      := 1,
           FBa                      := #xTmp,
           FBa2                     := I    274.6,
           Out                      := Q    274.6);

NETWORK
TITLE =SV_V1  Säurevorlaufventil Kreis 1
// Act 007
// Box           : VSRVK1..3
// Input address : I272.6
// Output address: Q272.6
      CALL FC    70 (
           UnitNo                   := #UnitNo,
           ActRec                   := DB2910.SV_V1,
           Typ                      := 1,
           FBa                      := #xTmp,
           FBa2                     := I    272.6,
           Out                      := Q    272.6);

NETWORK
TITLE =LV_V1  Laugevorlaufventil Kreis 1
// Act 008
// Box           : VSRVK1..3
// Input address : I272.3
// Output address: Q272.3
      CALL FC    70 (
           UnitNo                   := #UnitNo,
           ActRec                   := DB2910.LV_V1,
           Typ                      := 1,
           FBa                      := #xTmp,
           FBa2                     := I    272.3,
           Out                      := Q    272.3);

NETWORK
TITLE =LR_V1  Laugerücklaufventil Kreis 1
// Act 009
// Box           : VSRVK1..3
// Input address : I273.5
// Output address: Q273.5
      CALL FC    70 (
           UnitNo                   := #UnitNo,
           ActRec                   := DB2910.LR_V1,
           Typ                      := 1,
           FBa                      := #xTmp,
           FBa2                     := I    273.5,
           Out                      := Q    273.5);

NETWORK
TITLE =SR_V1  Säurerücklaufventil Kreis 1
// Act 010
// Box           : VSRVK1..3
// Input address : I274.0
// Output address: Q274.0
      CALL FC    70 (
           UnitNo                   := #UnitNo,
           ActRec                   := DB2910.SR_V1,
           Typ                      := 1,
           FBa                      := #xTmp,
           FBa2                     := I    274.0,
           Out                      := Q    274.0);

NETWORK
TITLE =HWR_V1  Heisswasserrücklaufventil Kreis 1
// Act 011
// Box           : VSRVK1..3
// Input address : I275.1
// Output address: Q275.1
      CALL FC    70 (
           UnitNo                   := #UnitNo,
           ActRec                   := DB2910.HWR_V1,
           Typ                      := 1,
           FBa                      := #xTmp,
           FBa2                     := I    275.1,
           Out                      := Q    275.1);

NETWORK
TITLE =GR_V1  Gullyventil Kreis 1
// Act 012
// Box           : VSRVK1..3
// Input address : I274.3
// Output address: Q274.3
      CALL FC    70 (
           UnitNo                   := #UnitNo,
           ActRec                   := DB2910.GR_V1,
           Typ                      := 1,
           FBa                      := #xTmp,
           FBa2                     := I    274.3,
           Out                      := Q    274.3);

NETWORK
TITLE =KV_V1  Kreislaufventil Kreis 1
// Act 032
// Box           : VSRVK1..3
// Input address : I272.0
// Output address: Q272.0
      CALL FC    70 (
           UnitNo                   := #UnitNo,
           ActRec                   := DB2910.KV_V1,
           Typ                      := 1,
           FBa                      := #xTmp,
           FBa2                     := I    272.0,
           Out                      := Q    272.0);

NETWORK
TITLE =CSRR1_MBU_A  Leitwertsonde Rücklauf Kontakt A (Lauge)
// Act 033
// Box           : S6 U6.3
// Output address: Q13.0
      CALL FC    70 (
           UnitNo                   := #UnitNo,
           ActRec                   := DB2910.CSRR1_MBU_A,
           Typ                      := 0,
           FBa                      := #xTmp,
           FBa2                     := #xTmp,
           Out                      := Q     13.0);

NETWORK
TITLE =CSRR1_MBU_B  Leitwertsonde Rücklauf Kontakt B (Saure)
// Act 034
// Box           : S6 U6.3
// Output address: Q13.1
      CALL FC    70 (
           UnitNo                   := #UnitNo,
           ActRec                   := DB2910.CSRR1_MBU_B,
           Typ                      := 0,
           FBa                      := #xTmp,
           FBa2                     := #xTmp,
           Out                      := Q     13.1);

END_FUNCTION_BLOCK

FUNCTION_BLOCK FB 1911
TITLE =U091: CIP Line 1
FAMILY : BOTEC_F1
NAME : UniE
VERSION : 1.2


VAR_TEMP
  CIP : BOOL ;	//CIP active
  UNIM : BOOL ;	//Unit Not In Maintenance
  GenRel : BOOL ;	//general OK (emergency and maintenance OK)
  EStopOK : BOOL ;	//emergency OK
  UnitNo : INT ;	//unit number
  xTmp : BOOL ;	//Temporary Bool
  iTmp : INT ;	//Temporary INT
  rTmp : REAL ;	//Temporary REAL
  dTmp : DINT ;	//Temporary DINT (free for general use)
  RetValInt : INT ;	//return value
END_VAR
BEGIN
NETWORK
TITLE =General

      SET   ;
// Simulation ---------------------------------------------------------------
      A     DB1911.DBX 1357.7;
      CC    FB  1919; // "U091Sim"
      A     DB1911.DBX   17.3;
      =     DB1911.DBX 1357.7; //Help bit for simulation

// get unit number ----------------------------------------------------------
      L     DB1910.DBW    0;
      T     #UnitNo;

// CIP ----------------------------------------------------------------------
      L     DB1911.DBD   54;
      L     0;
      <D    ;
      =     #CIP;

// emergency OK -------------------------------------------------------------
      A     DB1915.DBX   27.0; //Emergency Stop OK
      =     #EStopOK;

// Write Unit in Maintenance ------------------------------------------------

      AN    DB1911.DBX   69.7;
      =     #UNIM;

// emergency and maintenance OK ---------------------------------------------
      A     #EStopOK;
      A     #UNIM;
      =     #GenRel;

// communication ------------------------------------------------------------
      UC    FB  1915; // U091Com

NETWORK
TITLE =Sequence organisation

      CLR   ;
      =     M    122.2;

// SFM supply ----------------------------------------------------------------

// counter value to SFM DURCHFLUSSMESSUNG KREISLAUF 1 (U91) ----------------------
      CALL FC    44 (
           UnitNo                   := #UnitNo,
           CntRec                   := DB2912.IDM_IMPULSE_RV_1FQI,
           Enable                   := M     97.1,
           SFMRec                   := DB1911.Seq.SFM[14]);// Amount

// sequencer ----------------------------------------------------------------
      A     DB1913.DBX   43.1;
      S     DB1913.DBX   97.3;

      CALL FC    40 (
           UnitNo                   := #UnitNo);

END_FUNCTION_BLOCK

FUNCTION_BLOCK FB 1920
TITLE =U092: CIP Line 2
FAMILY : BOTEC_F1
NAME : UniA
VERSION : 2.1


VAR_TEMP
  EStopOK : BOOL ;	//auxiliary flag
  CIP : BOOL ;	//CIP Program Selected
  xTmp : BOOL ;	//Temporary Bool(free for general use)
  UnitNo : INT ;	//unit number
  UnitFB : INT ;	//unit expansion FB number
  rTmp : REAL ;	//Temporary REAL (free for general use)
  iTmp : INT ;	//Temporary INT (free for general use)
  dTmp : DINT ;	//Temporary DINT (free for general use)
END_VAR
BEGIN
NETWORK
TITLE =general

      CLR   ;
      =     #xTmp;
      =     #EStopOK;

      L     DB1920.DBW    0;
      T     #UnitNo;
      L     DB1920.DBW    2;
      T     #UnitFB;

NETWORK
TITLE =analog inputs

      NOP   0;
// RV2T1 AnI 001 Temperatur CIP Vorlauf 2
      CALL FC    24 (
           UnitNo                   := #UnitNo,
           AnIRec                   := DB2923.RV2T1,
           ValPer                   := IW   226);

// TI_RR2 AnI 002 Temperatur CIP Rücklauf 2
      CALL FC    24 (
           UnitNo                   := #UnitNo,
           AnIRec                   := DB2923.TI_RR2,
           ValPer                   := IW   136);

// CS_RR2 AnI 003 Leitwert CIP Rücklauf 2
      CALL FC    24 (
           UnitNo                   := #UnitNo,
           AnIRec                   := DB2923.CS_RR2,
           ValPer                   := IW   142);

// FIT_RV2 AnI 004 Flow CIP Kreislauf 2
      CALL FC    24 (
           UnitNo                   := #UnitNo,
           AnIRec                   := DB2923.FIT_RV2,
           ValPer                   := IW   130);

NETWORK
TITLE =Universal value

      NOP   0;
// unv001 UnV 001 Process Status
      CALL FC    27 (
           UnitNo                   := #UnitNo,
           UnVRec                   := DB2925.unv001,
           ValExt                   := DB2925.DBD  234);

// unv002 UnV 002 Universal Value 02
      CALL FC    27 (
           UnitNo                   := #UnitNo,
           UnVRec                   := DB2925.unv002,
           ValExt                   := DB2925.DBD  362);

NETWORK
TITLE =special inputs

      NOP   0;
// FS_RR2_NEU SpI 001
      CALL FC    14 (
           UnitNo                   := #UnitNo,
           SpIRec                   := DB2921.FS_RR2_NEU,
           SpIBit                   := I     94.1);

// IDM_IMPULSE_RV_2FQS SpI 002 DURCHFLUSSMESSUNG KREISLAUF 2
      CALL FC    14 (
           UnitNo                   := #UnitNo,
           SpIRec                   := DB2921.IDM_IMPULSE_RV_2FQS,
           SpIBit                   := I      0.1);

NETWORK
TITLE =messages

      NOP   0;
// msg001 Msg 001 Message 01
      CALL FC    16 (
           UnitNo                   := #UnitNo,
           MsgRec                   := DB2927.msg001,
           MsgBit                   := DB2927.DBX   82.7);

// msg002 Msg 002 Message 02
      CALL FC    16 (
           UnitNo                   := #UnitNo,
           MsgRec                   := DB2927.msg002,
           MsgBit                   := DB2927.DBX  142.7);

NETWORK
TITLE =counters

      NOP   0;
// IDM_IMPULSE_RV_2FQI Cnt 002 DURCHFLUSSMESSUNG KREISLAUF 2 (U92)
      CALL FC    25 (
           UnitNo                   := #UnitNo,
           CntRec                   := DB2922.IDM_IMPULSE_RV_2FQI,
           Imp                      := DB2922.DBX  179.0);

NETWORK
TITLE =controllers

      NOP   0;
// RV2RV PID 001 CIP 2
      CALL FC    55 (
           UnitNo                   := #UnitNo,
           PIDRec                   := DB2926.RV2RV,
           SpExt                    := DB2926.DBD  234,
           PVal                     := DB2926.DBD  254,
           OPer                     := QW   226);

NETWORK
TITLE =unit supply

      UC    FB [#UnitFB];

NETWORK
TITLE =RV_P2  Reinigungsvorlaufpumpe Kreis 2
// Act 001
// Box           : LT-CIP
// Input address : I256.1
// Output address: Q256.1
      CALL FC    70 (
           UnitNo                   := #UnitNo,
           ActRec                   := DB2920.RV_P2,
           Typ                      := 3,
           FBa                      := I    256.1,
           FBa2                     := #xTmp,
           Out                      := Q    256.1);

NETWORK
TITLE =RV2_RV  Regelventil CIP2
// Act 004
// Box           :
// Output address: #xTmp
      CALL FC    70 (
           UnitNo                   := #UnitNo,
           ActRec                   := DB2920.RV2_RV,
           Typ                      := 0,
           FBa                      := #xTmp,
           FBa2                     := #xTmp,
           Out                      := Q     14.2);

NETWORK
TITLE =FW_V2  Frischwasservorlaufventil Kreis 2
// Act 005
// Box           : VSRVK1..3
// Input address : I273.2
// Output address: Q273.2
      CALL FC    70 (
           UnitNo                   := #UnitNo,
           ActRec                   := DB2920.FW_V2,
           Typ                      := 1,
           FBa                      := #xTmp,
           FBa2                     := I    273.2,
           Out                      := Q    273.2);

NETWORK
TITLE =HW_V2  Heisswasservorlaufventil Kreis 2
// Act 006
// Box           : VSRVK1..3
// Input address : I274.7
// Output address: Q274.7
      CALL FC    70 (
           UnitNo                   := #UnitNo,
           ActRec                   := DB2920.HW_V2,
           Typ                      := 1,
           FBa                      := #xTmp,
           FBa2                     := I    274.7,
           Out                      := Q    274.7);

NETWORK
TITLE =SV_V2  Säurevorlaufventil Kreis 2
// Act 007
// Box           : VSRVK1..3
// Input address : I272.7
// Output address: Q272.7
      CALL FC    70 (
           UnitNo                   := #UnitNo,
           ActRec                   := DB2920.SV_V2,
           Typ                      := 1,
           FBa                      := #xTmp,
           FBa2                     := I    272.7,
           Out                      := Q    272.7);

NETWORK
TITLE =LV_V2  Laugevorlaufventil Kreis 2
// Act 008
// Box           : VSRVK1..3
// Input address : I272.4
// Output address: Q272.4
      CALL FC    70 (
           UnitNo                   := #UnitNo,
           ActRec                   := DB2920.LV_V2,
           Typ                      := 1,
           FBa                      := #xTmp,
           FBa2                     := I    272.4,
           Out                      := Q    272.4);

NETWORK
TITLE =LR_V2  Laugerücklaufventil Kreis 2
// Act 009
// Box           : VSRVK1..3
// Input address : I273.6
// Output address: Q273.6
      CALL FC    70 (
           UnitNo                   := #UnitNo,
           ActRec                   := DB2920.LR_V2,
           Typ                      := 1,
           FBa                      := #xTmp,
           FBa2                     := I    273.6,
           Out                      := Q    273.6);

NETWORK
TITLE =SR_V2  Säurerücklaufventil Kreis 2
// Act 010
// Box           : VSRVK1..3
// Input address : I274.1
// Output address: Q274.1
      CALL FC    70 (
           UnitNo                   := #UnitNo,
           ActRec                   := DB2920.SR_V2,
           Typ                      := 1,
           FBa                      := #xTmp,
           FBa2                     := I    274.1,
           Out                      := Q    274.1);

NETWORK
TITLE =HWR_V2  Heisswasserrücklaufventil Kreis 2
// Act 011
// Box           : VSRVK1..3
// Input address : I275.2
// Output address: Q275.2
      CALL FC    70 (
           UnitNo                   := #UnitNo,
           ActRec                   := DB2920.HWR_V2,
           Typ                      := 1,
           FBa                      := #xTmp,
           FBa2                     := I    275.2,
           Out                      := Q    275.2);

NETWORK
TITLE =GR_V2  Gullyventil Kreis 2
// Act 012
// Box           : VSRVK1..3
// Input address : I274.4
// Output address: Q274.4
      CALL FC    70 (
           UnitNo                   := #UnitNo,
           ActRec                   := DB2920.GR_V2,
           Typ                      := 1,
           FBa                      := #xTmp,
           FBa2                     := I    274.4,
           Out                      := Q    274.4);

NETWORK
TITLE =KV_V2  Kreislaufventil Kreis 2
// Act 032
// Box           : VSRVK1..3
// Input address : I272.1
// Output address: Q272.1
      CALL FC    70 (
           UnitNo                   := #UnitNo,
           ActRec                   := DB2920.KV_V2,
           Typ                      := 1,
           FBa                      := #xTmp,
           FBa2                     := I    272.1,
           Out                      := Q    272.1);

NETWORK
TITLE =CSRR2_MBU_A  Leitwertsonde Rücklauf2 Kontakt A (Lauge)
// Act 033
// Box           : S6 U6.3
// Output address: Q13.2
      CALL FC    70 (
           UnitNo                   := #UnitNo,
           ActRec                   := DB2920.CSRR2_MBU_A,
           Typ                      := 0,
           FBa                      := #xTmp,
           FBa2                     := #xTmp,
           Out                      := Q     13.2);

NETWORK
TITLE =CSRR2_MBU_B  Leitwertsonde Rücklauf2 Kontakt B (Saure)
// Act 034
// Box           : S6 U6.3
// Output address: Q13.3
      CALL FC    70 (
           UnitNo                   := #UnitNo,
           ActRec                   := DB2920.CSRR2_MBU_B,
           Typ                      := 0,
           FBa                      := #xTmp,
           FBa2                     := #xTmp,
           Out                      := Q     13.3);

END_FUNCTION_BLOCK

FUNCTION_BLOCK FB 1921
TITLE =U092: CIP Line 2
FAMILY : BOTEC_F1
NAME : UniE
VERSION : 1.2


VAR_TEMP
  CIP : BOOL ;	//CIP active
  UNIM : BOOL ;	//Unit Not In Maintenance
  GenRel : BOOL ;	//general OK (emergency and maintenance OK)
  EStopOK : BOOL ;	//emergency OK
  UnitNo : INT ;	//unit number
  xTmp : BOOL ;	//Temporary Bool
  iTmp : INT ;	//Temporary INT
  rTmp : REAL ;	//Temporary REAL
  dTmp : DINT ;	//Temporary DINT (free for general use)
  RetValInt : INT ;	//return value
END_VAR
BEGIN
NETWORK
TITLE =General

      SET   ;
// Simulation ---------------------------------------------------------------
      A     DB1921.DBX 1357.7;
      CC    FB  1929; // "U092Sim"
      A     DB1921.DBX   17.3;
      =     DB1921.DBX 1357.7; //Help bit for simulation

// get unit number ----------------------------------------------------------
      L     DB1920.DBW    0;
      T     #UnitNo;

// CIP ----------------------------------------------------------------------
      L     DB1921.DBD   54;
      L     0;
      <D    ;
      =     #CIP;

// emergency OK -------------------------------------------------------------
      A     DB1925.DBX   27.0; //Emergency Stop OK
      =     #EStopOK;

// Write Unit in Maintenance ------------------------------------------------

      AN    DB1921.DBX   69.7;
      =     #UNIM;

// emergency and maintenance OK ---------------------------------------------
      A     #EStopOK;
      A     #UNIM;
      =     #GenRel;

// communication ------------------------------------------------------------
      UC    FB  1925; // U092Com

NETWORK
TITLE =Sequence organisation

      CLR   ;
      =     M    122.2;

// SFM supply ----------------------------------------------------------------

// counter value to SFM DURCHFLUSSMESSUNG KREISLAUF 2 (U92) ----------------------
      CALL FC    44 (
           UnitNo                   := #UnitNo,
           CntRec                   := DB2922.IDM_IMPULSE_RV_2FQI,
           Enable                   := M     97.1,
           SFMRec                   := DB1921.Seq.SFM[14]);// Amount

// sequencer ----------------------------------------------------------------
      A     DB1923.DBX   43.1;
      S     DB1923.DBX   97.3;

      CALL FC    40 (
           UnitNo                   := #UnitNo);

END_FUNCTION_BLOCK

FUNCTION_BLOCK FB 1930
TITLE =U093: CIP Line 3
FAMILY : BOTEC_F1
NAME : UniA
VERSION : 2.1


VAR_TEMP
  EStopOK : BOOL ;	//auxiliary flag
  CIP : BOOL ;	//CIP Program Selected
  xTmp : BOOL ;	//Temporary Bool(free for general use)
  UnitNo : INT ;	//unit number
  UnitFB : INT ;	//unit expansion FB number
  rTmp : REAL ;	//Temporary REAL (free for general use)
  iTmp : INT ;	//Temporary INT (free for general use)
  dTmp : DINT ;	//Temporary DINT (free for general use)
END_VAR
BEGIN
NETWORK
TITLE =general

      CLR   ;
      =     #xTmp;
      =     #EStopOK;

      L     DB1930.DBW    0;
      T     #UnitNo;
      L     DB1930.DBW    2;
      T     #UnitFB;

NETWORK
TITLE =analog inputs

      NOP   0;
// RV3T1 AnI 001 Temperatur CIP Vorlauf 3
      CALL FC    24 (
           UnitNo                   := #UnitNo,
           AnIRec                   := DB2933.RV3T1,
           ValPer                   := IW   228);

// TI_RR3 AnI 002 Temperatur CIP Rücklauf 3
      CALL FC    24 (
           UnitNo                   := #UnitNo,
           AnIRec                   := DB2933.TI_RR3,
           ValPer                   := IW   138);

// CS_RR3 AnI 003 Leitwert CIP Rücklauf 3
      CALL FC    24 (
           UnitNo                   := #UnitNo,
           AnIRec                   := DB2933.CS_RR3,
           ValPer                   := IW   144);

// FIT_RV3 AnI 004 Flow CIP Kreislauf 3
      CALL FC    24 (
           UnitNo                   := #UnitNo,
           AnIRec                   := DB2933.FIT_RV3,
           ValPer                   := IW   132);

NETWORK
TITLE =Universal value

      NOP   0;
// unv001 UnV 001 Process Status
      CALL FC    27 (
           UnitNo                   := #UnitNo,
           UnVRec                   := DB2935.unv001,
           ValExt                   := DB2935.DBD  234);

// unv002 UnV 002 Universal Value 02
      CALL FC    27 (
           UnitNo                   := #UnitNo,
           UnVRec                   := DB2935.unv002,
           ValExt                   := DB2935.DBD  362);

NETWORK
TITLE =special inputs

      NOP   0;
// FS_RR3_ALT SpI 001 FS Reinigungsrücklauf
      CALL FC    14 (
           UnitNo                   := #UnitNo,
           SpIRec                   := DB2931.FS_RR3_ALT,
           SpIBit                   := I      7.5);

// IDM_IMPULSE_RV_3FQS SpI 002 DURCHFLUSSMESSUNG KREISLAUF 3
      CALL FC    14 (
           UnitNo                   := #UnitNo,
           SpIRec                   := DB2931.IDM_IMPULSE_RV_3FQS,
           SpIBit                   := I      0.2);

// FS_RR3_NEU SpI 003
//      CALL  "SI1"
//       UnitNo:=#UnitNo
//       SpIRec:="U093SpID".FS_RR3_NEU
//       SpIBit:="FS_RR3_NEU"


NETWORK
TITLE =messages

      NOP   0;
// msg001 Msg 001 Message 01
      CALL FC    16 (
           UnitNo                   := #UnitNo,
           MsgRec                   := DB2937.msg001,
           MsgBit                   := DB2937.DBX   82.7);

// msg002 Msg 002 Message 02
      CALL FC    16 (
           UnitNo                   := #UnitNo,
           MsgRec                   := DB2937.msg002,
           MsgBit                   := DB2937.DBX  142.7);

NETWORK
TITLE =counters

      NOP   0;
// IDM_IMPULSE_RV_3FQI Cnt 002 DURCHFLUSSMESSUNG KREISLAUF 3 (U93)
      CALL FC    25 (
           UnitNo                   := #UnitNo,
           CntRec                   := DB2932.IDM_IMPULSE_RV_3FQI,
           Imp                      := DB2932.DBX  179.0);

NETWORK
TITLE =controllers

      NOP   0;
// RV3RV PID 001 CIP 3
      CALL FC    55 (
           UnitNo                   := #UnitNo,
           PIDRec                   := DB2936.RV3RV,
           SpExt                    := DB2936.DBD  234,
           PVal                     := DB2936.DBD  254,
           OPer                     := QW   228);

NETWORK
TITLE =unit supply

      UC    FB [#UnitFB];

NETWORK
TITLE =RV_P3  RVP3 Reinigungsvorlaufpumpe Kreis 3
// Act 001
// Box           : S6 U6.3
// Input address : I5.7
// Output address: Q5.7
      CALL FC    70 (
           UnitNo                   := #UnitNo,
           ActRec                   := DB2930.RV_P3,
           Typ                      := 1,
           FBa                      := #xTmp,
           FBa2                     := I      5.7,
           Out                      := Q      5.7);

NETWORK
TITLE =RV3_RV  Regelventil CIP3
// Act 004
// Box           : ?
// Input address : #xTmp
// Output address: #xTmp
      CALL FC    70 (
           UnitNo                   := #UnitNo,
           ActRec                   := DB2930.RV3_RV,
           Typ                      := 0,
           FBa                      := #xTmp,
           FBa2                     := #xTmp,
           Out                      := Q     14.3);

NETWORK
TITLE =FW_V3  Frischwasservorlaufventil Kreis 3
// Act 005
// Box           : VSRVK1..3
// Input address : I273.3
// Output address: Q273.3
      CALL FC    70 (
           UnitNo                   := #UnitNo,
           ActRec                   := DB2930.FW_V3,
           Typ                      := 1,
           FBa                      := #xTmp,
           FBa2                     := I    273.3,
           Out                      := Q    273.3);

NETWORK
TITLE =HW_V3  Heisswasservorlaufventil Kreis 3
// Act 006
// Box           : VSRVK1..3
// Input address : I275.0
// Output address: Q275.0
      CALL FC    70 (
           UnitNo                   := #UnitNo,
           ActRec                   := DB2930.HW_V3,
           Typ                      := 1,
           FBa                      := #xTmp,
           FBa2                     := I    275.0,
           Out                      := Q    275.0);

NETWORK
TITLE =SV_V3  Säurevorlaufventil Kreis 3
// Act 007
// Box           : VSRVK1..3
// Input address : I273.0
// Output address: Q273.0
      CALL FC    70 (
           UnitNo                   := #UnitNo,
           ActRec                   := DB2930.SV_V3,
           Typ                      := 1,
           FBa                      := #xTmp,
           FBa2                     := I    273.0,
           Out                      := Q    273.0);

NETWORK
TITLE =LV_V3  Laugevorlaufventil Kreis 3
// Act 008
// Box           : VSRVK1..3
// Input address : I272.5
// Output address: Q272.5
      CALL FC    70 (
           UnitNo                   := #UnitNo,
           ActRec                   := DB2930.LV_V3,
           Typ                      := 1,
           FBa                      := #xTmp,
           FBa2                     := I    272.5,
           Out                      := Q    272.5);

NETWORK
TITLE =LR_V3  Laugerücklaufventil Kreis 3
// Act 009
// Box           : VSRVK1..3
// Input address : I273.7
// Output address: Q273.7
      CALL FC    70 (
           UnitNo                   := #UnitNo,
           ActRec                   := DB2930.LR_V3,
           Typ                      := 1,
           FBa                      := #xTmp,
           FBa2                     := I    273.7,
           Out                      := Q    273.7);

NETWORK
TITLE =SR_V3  Säurerücklaufventil Kreis 3
// Act 010
// Box           : VSRVK1..3
// Input address : I274.2
// Output address: Q274.2
      CALL FC    70 (
           UnitNo                   := #UnitNo,
           ActRec                   := DB2930.SR_V3,
           Typ                      := 1,
           FBa                      := #xTmp,
           FBa2                     := I    274.2,
           Out                      := Q    274.2);

NETWORK
TITLE =HWR_V3  Heisswasserrücklaufventil Kreis 3
// Act 011
// Box           : VSRVK1..3
// Input address : I275.3
// Output address: Q275.3
      CALL FC    70 (
           UnitNo                   := #UnitNo,
           ActRec                   := DB2930.HWR_V3,
           Typ                      := 1,
           FBa                      := #xTmp,
           FBa2                     := I    275.3,
           Out                      := Q    275.3);

NETWORK
TITLE =GR_V3  Gullyventil Kreis 3
// Act 012
// Box           : VSRVK1..3
// Input address : I274.5
// Output address: Q274.5
      CALL FC    70 (
           UnitNo                   := #UnitNo,
           ActRec                   := DB2930.GR_V3,
           Typ                      := 1,
           FBa                      := #xTmp,
           FBa2                     := I    274.5,
           Out                      := Q    274.5);

NETWORK
TITLE =KV_V3  Kreislaufventil Kreis 3
// Act 032
// Box           : VSRVK1..3
// Input address : I272.2
// Output address: Q272.2
      CALL FC    70 (
           UnitNo                   := #UnitNo,
           ActRec                   := DB2930.KV_V3,
           Typ                      := 1,
           FBa                      := #xTmp,
           FBa2                     := I    272.2,
           Out                      := Q    272.2);

NETWORK
TITLE =CSRR3_MBU_A  Leitwertsonde Rücklauf3 Kontakt A (Lauge)
// Act 033
// Box           : S6 U6.3
// Output address: Q13.4
      CALL FC    70 (
           UnitNo                   := #UnitNo,
           ActRec                   := DB2930.CSRR3_MBU_A,
           Typ                      := 0,
           FBa                      := #xTmp,
           FBa2                     := #xTmp,
           Out                      := Q     13.4);

NETWORK
TITLE =CSRR3_MBU_B  Leitwertsonde Rücklauf3 Kontakt B (Saure)
// Act 034
// Box           : S6 U6.3
// Output address: Q13.5
      CALL FC    70 (
           UnitNo                   := #UnitNo,
           ActRec                   := DB2930.CSRR3_MBU_B,
           Typ                      := 0,
           FBa                      := #xTmp,
           FBa2                     := #xTmp,
           Out                      := Q     13.5);

END_FUNCTION_BLOCK

FUNCTION_BLOCK FB 1931
TITLE =U093: CIP Line 3
FAMILY : BOTEC_F1
NAME : UniE
VERSION : 1.2


VAR_TEMP
  CIP : BOOL ;	//CIP active
  UNIM : BOOL ;	//Unit Not In Maintenance
  GenRel : BOOL ;	//general OK (emergency and maintenance OK)
  EStopOK : BOOL ;	//emergency OK
  UnitNo : INT ;	//unit number
  xTmp : BOOL ;	//Temporary Bool
  iTmp : INT ;	//Temporary INT
  rTmp : REAL ;	//Temporary REAL
  dTmp : DINT ;	//Temporary DINT (free for general use)
  RetValInt : INT ;	//return value
END_VAR
BEGIN
NETWORK
TITLE =General



      SET   ;
// Simulation ---------------------------------------------------------------
      A     DB1931.DBX 1357.7;
      CC    FB  1939; // "U093Sim"
      A     DB1931.DBX   17.3;
      =     DB1931.DBX 1357.7; //Help bit for simulation

// get unit number ----------------------------------------------------------
      L     DB1930.DBW    0;
      T     #UnitNo;

// CIP ----------------------------------------------------------------------
      L     DB1931.DBD   54;
      L     0;
      <D    ;
      =     #CIP;

// emergency OK -------------------------------------------------------------
      A     DB1935.DBX   27.0; //Emergency Stop OK
      =     #EStopOK;

// Write Unit in Maintenance ------------------------------------------------

      AN    DB1931.DBX   69.7;
      =     #UNIM;

// emergency and maintenance OK ---------------------------------------------
      A     #EStopOK;
      A     #UNIM;
      =     #GenRel;

// communication ------------------------------------------------------------
      UC    FB  1935; // U093Com

NETWORK
TITLE =Sequence organisation

      CLR   ;
      =     M    122.2;

// SFM supply ----------------------------------------------------------------

// counter value to SFM DURCHFLUSSMESSUNG KREISLAUF 3 (U93) ----------------------
      CALL FC    44 (
           UnitNo                   := #UnitNo,
           CntRec                   := DB2932.IDM_IMPULSE_RV_3FQI,
           Enable                   := M     97.1,
           SFMRec                   := DB1931.Seq.SFM[14]);// Amount

// sequencer ----------------------------------------------------------------
      A     DB1933.DBX   43.1;
      S     DB1933.DBX   97.3;

      CALL FC    40 (
           UnitNo                   := #UnitNo);

END_FUNCTION_BLOCK

FUNCTION_BLOCK FB 1940
TITLE =U094: CIP 1 Distribution
FAMILY : BOTEC_F1
NAME : UniA
VERSION : 2.1


VAR_TEMP
  EStopOK : BOOL ;	//auxiliary flag
  CIP : BOOL ;	//CIP Program Selected
  xTmp : BOOL ;	//Temporary Bool(free for general use)
  DummyBool : BOOL ;	//Temporary Bool(free for general use)
  UnitNo : INT ;	//unit number
  UnitFB : INT ;	//unit expansion FB number
  rTmp : REAL ;	//Temporary REAL (free for general use)
  iTmp : INT ;	//Temporary INT (free for general use)
  dTmp : DINT ;	//Temporary DINT (free for general use)
END_VAR
BEGIN
NETWORK
TITLE =general

      CLR   ;
      =     #xTmp;
      =     #EStopOK;

      L     DB1940.DBW    0;
      T     #UnitNo;
      L     DB1940.DBW    2;
      T     #UnitFB;

NETWORK
TITLE =Universal value

      NOP   0;
// unv001 UnV 001 Process Status
      CALL FC    27 (
           UnitNo                   := #UnitNo,
           UnVRec                   := DB2945.unv001,
           ValExt                   := DB2945.DBD  234);

// unv002 UnV 002 Universal Value 02
      CALL FC    27 (
           UnitNo                   := #UnitNo,
           UnVRec                   := DB2945.unv002,
           ValExt                   := DB2945.DBD  362);

// RK1_KreisNr UnV 003 Circuit Number
      CALL FC    27 (
           UnitNo                   := #UnitNo,
           UnVRec                   := DB2945.RK1_KreisNr,
           ValExt                   := DB2945.DBD  490);

// RK1_Medium UnV 004 0=NIX 1=Wasser 2=Heißwasser 3=Lauge 4=Säure 5=Desi
      CALL FC    27 (
           UnitNo                   := #UnitNo,
           UnVRec                   := DB2945.RK1_Medium,
           ValExt                   := DB2945.DBD  618);

NETWORK
TITLE =special inputs

      NOP   0;
// RK1_I_Bereit SpI 001 Das Reinigungs Programm ist gestartet und läuft "1"= Läuft  "0"=AUS
      CALL FC    14 (
           UnitNo                   := #UnitNo,
           SpIRec                   := DB2941.RK1_I_Bereit,
           SpIBit                   := DB304.DBX   10.0);

// RK1_I_VL_Ein SpI 002 Medium wird angefordert (Reinigungs Vorlauf EIN) "1"=VorlaufPumpe an "0"AUS
      CALL FC    14 (
           UnitNo                   := #UnitNo,
           SpIRec                   := DB2941.RK1_I_VL_Ein,
           SpIBit                   := DB304.DBX   10.1);

// RK1_I_RL_Ein SpI 003 Medium wird zurückgepumpt "1" RücklaufPumpe an "0"=AUS
      CALL FC    14 (
           UnitNo                   := #UnitNo,
           SpIRec                   := DB2941.RK1_I_RL_Ein,
           SpIBit                   := DB304.DBX   10.2);

// RK1_I_Leer SpI 004 Der zu Reinigende Anlagenteil ist leer."1"=leer "0"=nicht leer
      CALL FC    14 (
           UnitNo                   := #UnitNo,
           SpIRec                   := DB2941.RK1_I_Leer,
           SpIBit                   := DB304.DBX   10.3);

// RK1_I_Stop SpI 005 Stop interner Fehler Pumpen anhalten Reinigungszeit anhalten "1" STOP  "0"= OK
      CALL FC    14 (
           UnitNo                   := #UnitNo,
           SpIRec                   := DB2941.RK1_I_Stop,
           SpIBit                   := DB304.DBX   10.4);

// RK1_I_SK_RM SpI 006 Bypassventil ist angesteuert und offen
      CALL FC    14 (
           UnitNo                   := #UnitNo,
           SpIRec                   := DB2941.RK1_I_SK_RM,
           SpIBit                   := DB304.DBX   10.7);

NETWORK
TITLE =messages

      NOP   0;
// msg001 Msg 001 Message 01
      CALL FC    16 (
           UnitNo                   := #UnitNo,
           MsgRec                   := DB2947.msg001,
           MsgBit                   := DB2947.DBX   82.7);

// msg002 Msg 002 Message 02
      CALL FC    16 (
           UnitNo                   := #UnitNo,
           MsgRec                   := DB2947.msg002,
           MsgBit                   := DB2947.DBX  142.7);

NETWORK
TITLE =unit supply

      UC    FB [#UnitFB];

NETWORK
TITLE =RR_P1  RRP1 Reinigungsrücklaufpumpe Kreis 1
// Act 001
// Box           : S6 U6.3
// Input address : I6.6
// Output address: Q6.6
      CALL FC    70 (
           UnitNo                   := #UnitNo,
           ActRec                   := DB2940.RR_P1,
           Typ                      := 1,
           FBa                      := #xTmp,
           FBa2                     := I      6.6,
           Out                      := Q      6.6);

NETWORK
TITLE =U94_Act004  spare
// Act 004
// Box           :
// Output address: #DummyBool
      CALL FC    70 (
           UnitNo                   := #UnitNo,
           ActRec                   := DB2940.U94_Act004,
           Typ                      := 0,
           FBa                      := #xTmp,
           FBa2                     := #xTmp,
           Out                      := #DummyBool);

NETWORK
TITLE =KZE5_Ventil_zum_SR_auf  KZE5 Ventil zum Sirupraum öffnen V720085
// Act 005
// Box           : KZE5
// Input address: I347.0
// Output address: Q346.0
      CALL FC    70 (
           UnitNo                   := #UnitNo,
           ActRec                   := DB2940.KZE5_Ventil_zum_SR_auf,
           Typ                      := 3,
           FBa                      := I    347.0,
           FBa2                     := #xTmp,
           Out                      := Q    346.0);

NETWORK
TITLE =RR1_V2
// Act 006
// Box           : VSRVK1..3
// Input address : I82.3
// Output address: Q82.3
      CALL FC    70 (
           UnitNo                   := #UnitNo,
           ActRec                   := DB2940.RR1_V2,
           Typ                      := 1,
           FBa                      := #xTmp,
           FBa2                     := I     82.3,
           Out                      := Q     82.3);

NETWORK
TITLE =RR1_V3  Ventil CIP 1 -> KF
// Act 007
// Box           : VSRR1-3
// Input address : I85.7
// Output address: Q85.7
      CALL FC    70 (
           UnitNo                   := #UnitNo,
           ActRec                   := DB2940.RR1_V3,
           Typ                      := 1,
           FBa                      := #xTmp,
           FBa2                     := I     85.7,
           Out                      := Q     85.7);

NETWORK
TITLE =RV1_SK
// Act 008
// Box           : VSRVK1..3
// Input address : I82.0
// Output address: Q82.0
      CALL FC    70 (
           UnitNo                   := #UnitNo,
           ActRec                   := DB2940.RV1_SK,
           Typ                      := 1,
           FBa                      := #xTmp,
           FBa2                     := I     82.0,
           Out                      := Q     82.0);

NETWORK
TITLE =FW_RK1
// Act 009
// Box           : Ventilinsel 4
// Input address : I335.7
// Output address: Q335.7
//      CALL  "Act"
//       UnitNo:=#UnitNo
//       ActRec:="U094ActD".U094_Act009
//       Typ   :=0
//       FBa   :=#xTmp
//       FBa2  :="FW_RK1GSC"
//       Out   :="FW_RK1O"

NETWORK
TITLE =RK1_Bereit  Die CIP Station hat gestatet "0"=AUS "1"=gestartet
// Act 010
// Box           : Sirup
// Output address: DB_SEND_DOEHLER.RK1.Bereit
      CALL FC    70 (
           UnitNo                   := #UnitNo,
           ActRec                   := DB2940.RK1_Bereit,
           Typ                      := 0,
           FBa                      := #xTmp,
           FBa2                     := #xTmp,
           Out                      := DB404.DBX   10.0);

NETWORK
TITLE =RK1_Stop  Stop Pumpen anhalten "0"Ok" 1"=Stop
// Act 011
// Box           : Sirup
// Output address: DB_SEND_DOEHLER.RK1.Stop
      CALL FC    70 (
           UnitNo                   := #UnitNo,
           ActRec                   := DB2940.RK1_Stop,
           Typ                      := 0,
           FBa                      := #xTmp,
           FBa2                     := #xTmp,
           Out                      := DB404.DBX   10.1);

NETWORK
TITLE =RK1_MED  Medienwechsel der CIP
// Act 012
// Box           : Sirup
// Output address: DB_SEND_DOEHLER.RK1.MED
      CALL FC    70 (
           UnitNo                   := #UnitNo,
           ActRec                   := DB2940.RK1_MED,
           Typ                      := 0,
           FBa                      := #xTmp,
           FBa2                     := #xTmp,
           Out                      := DB404.DBX   10.2);

NETWORK
TITLE =RK1_ENDE  Ende der Reinigung
// Act 013
// Box           : Sirup
// Output address: DB_SEND_DOEHLER.RK1.ENDE
      CALL FC    70 (
           UnitNo                   := #UnitNo,
           ActRec                   := DB2940.RK1_ENDE,
           Typ                      := 0,
           FBa                      := #xTmp,
           FBa2                     := #xTmp,
           Out                      := DB404.DBX   10.3);

NETWORK
TITLE =RK1_Bypass  CIP Bypass
// Act 014
// Box           : Sirup
// Output address: DB_SEND_DOEHLER.RK1.Bypass
      CALL FC    70 (
           UnitNo                   := #UnitNo,
           ActRec                   := DB2940.RK1_Bypass,
           Typ                      := 0,
           FBa                      := #xTmp,
           FBa2                     := #xTmp,
           Out                      := DB404.DBX   10.4);

NETWORK
TITLE =SR1_RR1  SR1 RR1 CIP Rücklaufventil RR1SR1
// Act 015
// Box           : VS-RRA
// Input address : I200.6
// Output address: Q200.6
      CALL FC    70 (
           UnitNo                   := #UnitNo,
           ActRec                   := DB2940.SR1_RR1,
           Typ                      := 1,
           FBa                      := #xTmp,
           FBa2                     := I    200.6,
           Out                      := Q    200.6);

NETWORK
TITLE =SR2_RR1  SR2 RR1 CIP Rücklaufventil RR1SR2
// Act 016
// Box           : VS-RRA
// Input address : I201.0
// Output address: Q201.0
      CALL FC    70 (
           UnitNo                   := #UnitNo,
           ActRec                   := DB2940.SR2_RR1,
           Typ                      := 1,
           FBa                      := #xTmp,
           FBa2                     := I    201.0,
           Out                      := Q    201.0);

NETWORK
TITLE =RV1_T
// Act 017
// Box           : Ventilinsel 4
// Input address : I335.6
// Output address: Q335.6
      CALL FC    70 (
           UnitNo                   := #UnitNo,
           ActRec                   := DB2940.RV1_T,
           Typ                      := 1,
           FBa                      := #xTmp,
           FBa2                     := I    335.6,
           Out                      := Q    335.6);

NETWORK
TITLE =RV1_RR1
// Act 018
// Box           : Ventilinsel 4
// Input address : I335.5
// Output address: Q335.5
      CALL FC    70 (
           UnitNo                   := #UnitNo,
           ActRec                   := DB2940.RV1_RR1,
           Typ                      := 1,
           FBa                      := #xTmp,
           FBa2                     := I    335.5,
           Out                      := Q    335.5);

NETWORK
TITLE =RV1_RS  Ventil zum Gully beim spülen vom Tank
// Act 019
// Box           : Ventilinsel 4
// Input address : I337.2
// Output address: Q337.2
      CALL FC    70 (
           UnitNo                   := #UnitNo,
           ActRec                   := DB2940.RV1_RS,
           Typ                      := 1,
           FBa                      := #xTmp,
           FBa2                     := I    337.2,
           Out                      := Q    337.2);

END_FUNCTION_BLOCK

FUNCTION_BLOCK FB 1941
TITLE =U094: CIP 1 Distribution
FAMILY : BOTEC_F1
NAME : UniE
VERSION : 1.2


VAR_TEMP
  CIP : BOOL ;	//CIP active
  UNIM : BOOL ;	//Unit Not In Maintenance
  GenRel : BOOL ;	//general OK (emergency and maintenance OK)
  EStopOK : BOOL ;	//emergency OK
  UnitNo : INT ;	//unit number
  xTmp : BOOL ;	//Temporary Bool
  iTmp : INT ;	//Temporary INT
  rTmp : REAL ;	//Temporary REAL
  dTmp : DINT ;	//Temporary DINT (free for general use)
  RetValInt : INT ;	//return value
END_VAR
BEGIN
NETWORK
TITLE =General

      SET   ;
// Simulation ---------------------------------------------------------------
      A     DB1941.DBX 1357.7;
      CC    FB  1949; // "U094Sim"
      A     DB1941.DBX   17.3;
      =     DB1941.DBX 1357.7; //Help bit for simulation

// get unit number ----------------------------------------------------------
      L     DB1940.DBW    0;
      T     #UnitNo;

// CIP ----------------------------------------------------------------------
      L     DB1941.DBD   54;
      L     0;
      <D    ;
      =     #CIP;

// emergency OK -------------------------------------------------------------
      A     DB1945.DBX   27.0; //Emergency Stop OK
      =     #EStopOK;

// Write Unit in Maintenance ------------------------------------------------

      AN    DB1941.DBX   69.7;
      =     #UNIM;

// emergency and maintenance OK ---------------------------------------------
      A     #EStopOK;
      A     #UNIM;
      =     #GenRel;

// communication ------------------------------------------------------------
      UC    FB  1945; // U094Com

NETWORK
TITLE =Universal Value

      NOP   0;

// ----------------------------------------------------------
// unv001 Process Status
// ----------------------------------------------------------
// process value to UnV
//      L     0.000000e+000
//      T     "U094UnVD".unv001.ValExt

// ----------------------------------------------------------
// unv002 Universal Value 02
// ----------------------------------------------------------
// process value to UnV
//      L     0.000000e+000
//      T     "U094UnVD".unv002.ValExt

// ----------------------------------------------------------
// RK1_KreisNr Circuit Number
// ----------------------------------------------------------
// process value to UnV
//      L     0.000000e+000
//      T     "U094UnVD".RK1_KreisNr.ValExt

// ----------------------------------------------------------
// RK1_Medium 0=NIX 1=Wasser 2=Heißwasser 3=Lauge 4=Säure 5=Desi
// ----------------------------------------------------------
// process value to UnV
//      L     0.000000e+000
//      T     "U094UnVD".RK1_Medium.ValExt

NETWORK
TITLE =Special Input

      NOP   0;

// ----------------------------------------------------------
// RK1_I_Bereit Das Reinigungs Programm ist gestartet und läuft "1"= Läuft  "0"=AUS
// ----------------------------------------------------------
      CLR   ;
      =     DB2941.DBX   81.4;
      =     DB2941.DBX   81.5;

// ----------------------------------------------------------
// RK1_I_VL_Ein Medium wird angefordert (Reinigungs Vorlauf EIN) "1"=VorlaufPumpe an "0"AUS
// ----------------------------------------------------------
      CLR   ;
      =     DB2941.DBX  141.4;
      =     DB2941.DBX  141.5;

// ----------------------------------------------------------
// RK1_I_RL_Ein Medium wird zurückgepumpt "1" RücklaufPumpe an "0"=AUS
// ----------------------------------------------------------
      CLR   ;
      =     DB2941.DBX  201.4;
      =     DB2941.DBX  201.5;

// ----------------------------------------------------------
// RK1_I_Leer Der zu Reinigende Anlagenteil ist leer."1"=leer "0"=nicht leer
// ----------------------------------------------------------
      CLR   ;
      =     DB2941.DBX  261.4;
      =     DB2941.DBX  261.5;

// ----------------------------------------------------------
// RK1_I_Stop Stop interner Fehler Pumpen anhalten Reinigungszeit anhalten "1" STOP  "0"= OK
// ----------------------------------------------------------
      CLR   ;
      =     DB2941.DBX  321.4;
      =     DB2941.DBX  321.5;

// ----------------------------------------------------------
// RK1_I_SK_RM Bypassventil ist angesteuert und offen
// ----------------------------------------------------------
      CLR   ;
      =     DB2941.DBX  381.4;
      =     DB2941.DBX  381.5;

NETWORK
TITLE =Messages

      NOP   0;

// ----------------------------------------------------------
// msg001 Message 01
// ----------------------------------------------------------
      SET   ;
      R     DB2947.DBX   80.7;
      =     DB2947.DBX   81.4;

      CLR   ;
      =     DB2947.DBX   82.7;

// ----------------------------------------------------------
// msg002 Message 02
// ----------------------------------------------------------
      SET   ;
      R     DB2947.DBX  140.7;
      =     DB2947.DBX  141.4;

      CLR   ;
      =     DB2947.DBX  142.7;

NETWORK
TITLE =Sequence organisation

      CLR   ;
      =     M    122.2;

// SFM supply ----------------------------------------------------------------

// CIP Counter
      CALL FC    29 (
           UnitNo                   := #UnitNo,
           Value                    := DB1945.DBD   54,
           Enable                   := TRUE,
           Down                     := FALSE,
           OriginDetect             := 0.000000e+000,
           MaxDiffPS                := 1.000000e+000,
           SFMRec                   := DB1941.Seq.SFM[15],
           ValueOld                 := DB1941.DBD 1418);

// sequencer ----------------------------------------------------------------
      A     DB1943.DBX   43.1;
      S     DB1943.DBX   97.3;

      CALL FC    40 (
           UnitNo                   := #UnitNo);

NETWORK
TITLE =Auto / Manual

      SET   ;
      AN    M    122.2;
      JC    MODE;
      AN    M    120.1;

// assign actuator mode
      AN    M    120.1;
      =     DB2940.DBX  105.4;
      =     DB2940.DBX  265.4;
      =     DB2940.DBX  345.4;
      =     DB2940.DBX  425.4;
      =     DB2940.DBX  505.4;
      =     DB2940.DBX  585.4;
      =     DB2940.DBX  665.4;
      =     DB2940.DBX  745.4;
      =     DB2940.DBX  825.4;
      =     DB2940.DBX  905.4;
      =     DB2940.DBX  985.4;
      =     DB2940.DBX 1065.4;
      =     DB2940.DBX 1145.4;
      =     DB2940.DBX 1225.4;
      =     DB2940.DBX 1305.4;
      =     DB2940.DBX 1385.4;
      =     DB2940.DBX 1465.4;
      =     DB2940.DBX 1545.4;



MODE: SET   ;

NETWORK
TITLE =RR_P1 RRP1 Reinigungsrücklaufpumpe Kreis 1
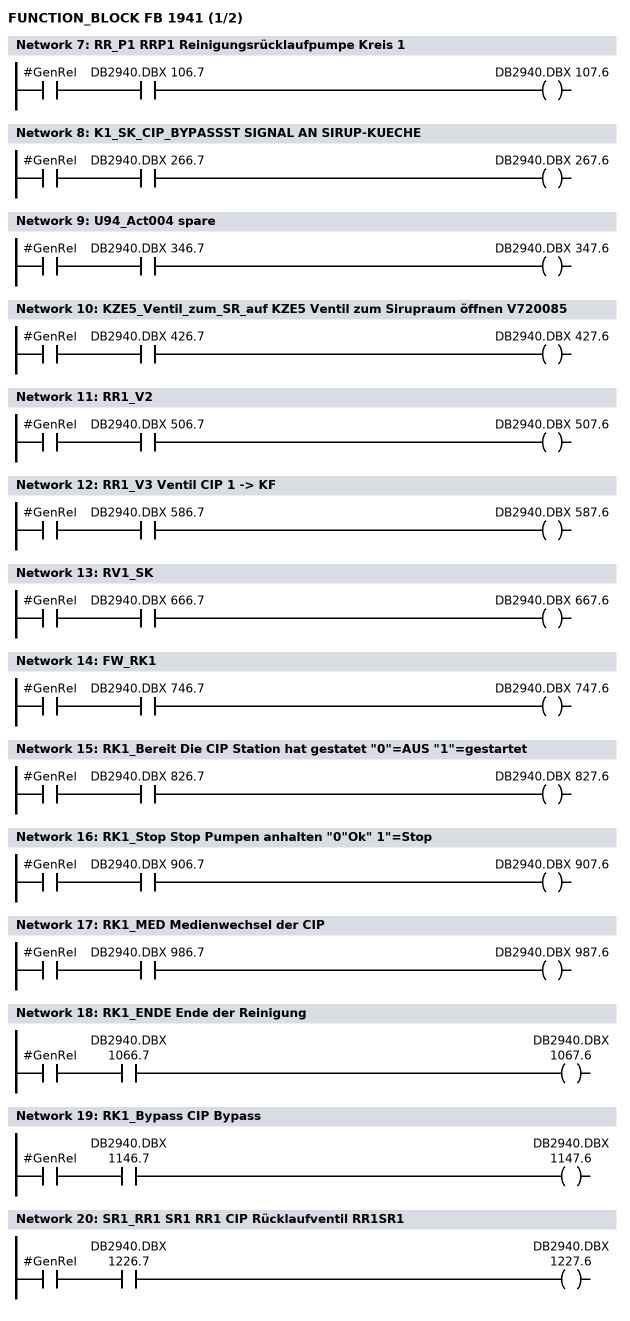

      A     #GenRel;
      A     DB2940.DBX  106.7;
      =     DB2940.DBX  107.6;
NETWORK
TITLE =K1_SK_CIP_BYPASSST SIGNAL AN SIRUP-KUECHE

      A     #GenRel;
      A     DB2940.DBX  266.7;
      =     DB2940.DBX  267.6;
NETWORK
TITLE =U94_Act004 spare

      A     #GenRel;
      A     DB2940.DBX  346.7;
      =     DB2940.DBX  347.6;
NETWORK
TITLE =KZE5_Ventil_zum_SR_auf KZE5 Ventil zum Sirupraum öffnen V720085

      A     #GenRel;
      A     DB2940.DBX  426.7;
      =     DB2940.DBX  427.6;
NETWORK
TITLE =RR1_V2

      A     #GenRel;
      A     DB2940.DBX  506.7;
      =     DB2940.DBX  507.6;
NETWORK
TITLE =RR1_V3 Ventil CIP 1 -> KF

      A     #GenRel;
      A     DB2940.DBX  586.7;
      =     DB2940.DBX  587.6;
NETWORK
TITLE =RV1_SK

      A     #GenRel;
      A     DB2940.DBX  666.7;
      =     DB2940.DBX  667.6;
NETWORK
TITLE =FW_RK1

      A     #GenRel;
      A     DB2940.DBX  746.7;
      =     DB2940.DBX  747.6;
NETWORK
TITLE =RK1_Bereit Die CIP Station hat gestatet "0"=AUS "1"=gestartet

      A     #GenRel;
      A     DB2940.DBX  826.7;
      =     DB2940.DBX  827.6;
NETWORK
TITLE =RK1_Stop Stop Pumpen anhalten "0"Ok" 1"=Stop

      A     #GenRel;
      A     DB2940.DBX  906.7;
      =     DB2940.DBX  907.6;
NETWORK
TITLE =RK1_MED Medienwechsel der CIP

      A     #GenRel;
      A     DB2940.DBX  986.7;
      =     DB2940.DBX  987.6;
NETWORK
TITLE =RK1_ENDE Ende der Reinigung

      A     #GenRel;
      A     DB2940.DBX 1066.7;
      =     DB2940.DBX 1067.6;
NETWORK
TITLE =RK1_Bypass CIP Bypass

      A     #GenRel;
      A     DB2940.DBX 1146.7;
      =     DB2940.DBX 1147.6;
NETWORK
TITLE =SR1_RR1 SR1 RR1 CIP Rücklaufventil RR1SR1

      A     #GenRel;
      A     DB2940.DBX 1226.7;
      =     DB2940.DBX 1227.6;
NETWORK
TITLE =SR2_RR1 SR2 RR1 CIP Rücklaufventil RR1SR2
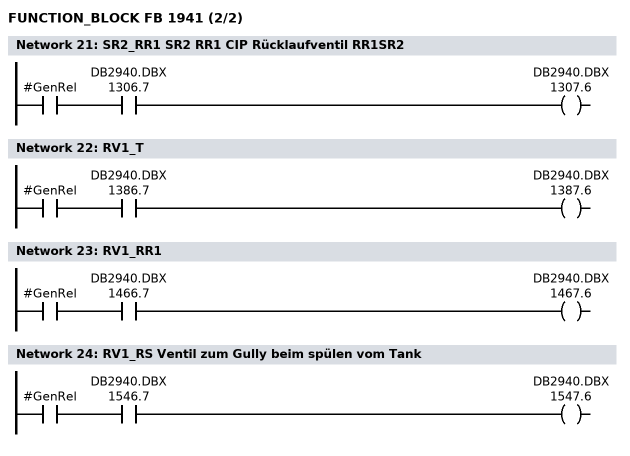

      A     #GenRel;
      A     DB2940.DBX 1306.7;
      =     DB2940.DBX 1307.6;
NETWORK
TITLE =RV1_T

      A     #GenRel;
      A     DB2940.DBX 1386.7;
      =     DB2940.DBX 1387.6;
NETWORK
TITLE =RV1_RR1

      A     #GenRel;
      A     DB2940.DBX 1466.7;
      =     DB2940.DBX 1467.6;
NETWORK
TITLE =RV1_RS Ventil zum Gully beim spülen vom Tank

      A     #GenRel;
      A     DB2940.DBX 1546.7;
      =     DB2940.DBX 1547.6;
END_FUNCTION_BLOCK

FUNCTION_BLOCK FB 1950
TITLE =U095: CIP 2 Distribution
FAMILY : BOTEC_F1
NAME : UniA
VERSION : 2.1


